# B&R Automation Studio project TD52 (part 15)

```c
/* Source: ctrttf.f */
#define ctrttf FORTRAN_WRAPPER(ctrttf)
extern void ctrttf(
    char   *transr,
    char   *uplo,
    ptrdiff_t *n,
    float  *a,
    ptrdiff_t *lda,
    float  *arf,
    ptrdiff_t *info
);

/* Source: ctrttp.f */
#define ctrttp FORTRAN_WRAPPER(ctrttp)
extern void ctrttp(
    char   *uplo,
    ptrdiff_t *n,
    float  *a,
    ptrdiff_t *lda,
    float  *ap,
    ptrdiff_t *info
);

/* Source: ctzrqf.f */
#define ctzrqf FORTRAN_WRAPPER(ctzrqf)
extern void ctzrqf(
    ptrdiff_t *m,
    ptrdiff_t *n,
    float  *a,
    ptrdiff_t *lda,
    float  *tau,
    ptrdiff_t *info
);

/* Source: ctzrzf.f */
#define ctzrzf FORTRAN_WRAPPER(ctzrzf)
extern void ctzrzf(
    ptrdiff_t *m,
    ptrdiff_t *n,
    float  *a,
    ptrdiff_t *lda,
    float  *tau,
    float  *work,
    ptrdiff_t *lwork,
    ptrdiff_t *info
);

/* Source: cung2l.f */
#define cung2l FORTRAN_WRAPPER(cung2l)
extern void cung2l(
    ptrdiff_t *m,
    ptrdiff_t *n,
    ptrdiff_t *k,
    float  *a,
    ptrdiff_t *lda,
    float  *tau,
    float  *work,
    ptrdiff_t *info
);

/* Source: cung2r.f */
#define cung2r FORTRAN_WRAPPER(cung2r)
extern void cung2r(
    ptrdiff_t *m,
    ptrdiff_t *n,
    ptrdiff_t *k,
    float  *a,
    ptrdiff_t *lda,
    float  *tau,
    float  *work,
    ptrdiff_t *info
);

/* Source: cungbr.f */
#define cungbr FORTRAN_WRAPPER(cungbr)
extern void cungbr(
    char   *vect,
    ptrdiff_t *m,
    ptrdiff_t *n,
    ptrdiff_t *k,
    float  *a,
    ptrdiff_t *lda,
    float  *tau,
    float  *work,
    ptrdiff_t *lwork,
    ptrdiff_t *info
);

/* Source: cunghr.f */
#define cunghr FORTRAN_WRAPPER(cunghr)
extern void cunghr(
    ptrdiff_t *n,
    ptrdiff_t *ilo,
    ptrdiff_t *ihi,
    float  *a,
    ptrdiff_t *lda,
    float  *tau,
    float  *work,
    ptrdiff_t *lwork,
    ptrdiff_t *info
);

/* Source: cungl2.f */
#define cungl2 FORTRAN_WRAPPER(cungl2)
extern void cungl2(
    ptrdiff_t *m,
    ptrdiff_t *n,
    ptrdiff_t *k,
    float  *a,
    ptrdiff_t *lda,
    float  *tau,
    float  *work,
    ptrdiff_t *info
);

/* Source: cunglq.f */
#define cunglq FORTRAN_WRAPPER(cunglq)
extern void cunglq(
    ptrdiff_t *m,
    ptrdiff_t *n,
    ptrdiff_t *k,
    float  *a,
    ptrdiff_t *lda,
    float  *tau,
    float  *work,
    ptrdiff_t *lwork,
    ptrdiff_t *info
);

/* Source: cungql.f */
#define cungql FORTRAN_WRAPPER(cungql)
extern void cungql(
    ptrdiff_t *m,
    ptrdiff_t *n,
    ptrdiff_t *k,
    float  *a,
    ptrdiff_t *lda,
    float  *tau,
    float  *work,
    ptrdiff_t *lwork,
    ptrdiff_t *info
);

/* Source: cungqr.f */
#define cungqr FORTRAN_WRAPPER(cungqr)
extern void cungqr(
    ptrdiff_t *m,
    ptrdiff_t *n,
    ptrdiff_t *k,
    float  *a,
    ptrdiff_t *lda,
    float  *tau,
    float  *work,
    ptrdiff_t *lwork,
    ptrdiff_t *info
);

/* Source: cungr2.f */
#define cungr2 FORTRAN_WRAPPER(cungr2)
extern void cungr2(
    ptrdiff_t *m,
    ptrdiff_t *n,
    ptrdiff_t *k,
    float  *a,
    ptrdiff_t *lda,
    float  *tau,
    float  *work,
    ptrdiff_t *info
);

/* Source: cungrq.f */
#define cungrq FORTRAN_WRAPPER(cungrq)
extern void cungrq(
    ptrdiff_t *m,
    ptrdiff_t *n,
    ptrdiff_t *k,
    float  *a,
    ptrdiff_t *lda,
    float  *tau,
    float  *work,
    ptrdiff_t *lwork,
    ptrdiff_t *info
);

/* Source: cungtr.f */
#define cungtr FORTRAN_WRAPPER(cungtr)
extern void cungtr(
    char   *uplo,
    ptrdiff_t *n,
    float  *a,
    ptrdiff_t *lda,
    float  *tau,
    float  *work,
    ptrdiff_t *lwork,
    ptrdiff_t *info
);

/* Source: cunm2l.f */
#define cunm2l FORTRAN_WRAPPER(cunm2l)
extern void cunm2l(
    char   *side,
    char   *trans,
    ptrdiff_t *m,
    ptrdiff_t *n,
    ptrdiff_t *k,
    float  *a,
    ptrdiff_t *lda,
    float  *tau,
    float  *c,
    ptrdiff_t *ldc,
    float  *work,
    ptrdiff_t *info
);

/* Source: cunm2r.f */
#define cunm2r FORTRAN_WRAPPER(cunm2r)
extern void cunm2r(
    char   *side,
    char   *trans,
    ptrdiff_t *m,
    ptrdiff_t *n,
    ptrdiff_t *k,
    float  *a,
    ptrdiff_t *lda,
    float  *tau,
    float  *c,
    ptrdiff_t *ldc,
    float  *work,
    ptrdiff_t *info
);

/* Source: cunmbr.f */
#define cunmbr FORTRAN_WRAPPER(cunmbr)
extern void cunmbr(
    char   *vect,
    char   *side,
    char   *trans,
    ptrdiff_t *m,
    ptrdiff_t *n,
    ptrdiff_t *k,
    float  *a,
    ptrdiff_t *lda,
    float  *tau,
    float  *c,
    ptrdiff_t *ldc,
    float  *work,
    ptrdiff_t *lwork,
    ptrdiff_t *info
);

/* Source: cunmhr.f */
#define cunmhr FORTRAN_WRAPPER(cunmhr)
extern void cunmhr(
    char   *side,
    char   *trans,
    ptrdiff_t *m,
    ptrdiff_t *n,
    ptrdiff_t *ilo,
    ptrdiff_t *ihi,
    float  *a,
    ptrdiff_t *lda,
    float  *tau,
    float  *c,
    ptrdiff_t *ldc,
    float  *work,
    ptrdiff_t *lwork,
    ptrdiff_t *info
);

/* Source: cunml2.f */
#define cunml2 FORTRAN_WRAPPER(cunml2)
extern void cunml2(
    char   *side,
    char   *trans,
    ptrdiff_t *m,
    ptrdiff_t *n,
    ptrdiff_t *k,
    float  *a,
    ptrdiff_t *lda,
    float  *tau,
    float  *c,
    ptrdiff_t *ldc,
    float  *work,
    ptrdiff_t *info
);

/* Source: cunmlq.f */
#define cunmlq FORTRAN_WRAPPER(cunmlq)
extern void cunmlq(
    char   *side,
    char   *trans,
    ptrdiff_t *m,
    ptrdiff_t *n,
    ptrdiff_t *k,
    float  *a,
    ptrdiff_t *lda,
    float  *tau,
    float  *c,
    ptrdiff_t *ldc,
    float  *work,
    ptrdiff_t *lwork,
    ptrdiff_t *info
);

/* Source: cunmql.f */
#define cunmql FORTRAN_WRAPPER(cunmql)
extern void cunmql(
    char   *side,
    char   *trans,
    ptrdiff_t *m,
    ptrdiff_t *n,
    ptrdiff_t *k,
    float  *a,
    ptrdiff_t *lda,
    float  *tau,
    float  *c,
    ptrdiff_t *ldc,
    float  *work,
    ptrdiff_t *lwork,
    ptrdiff_t *info
);

/* Source: cunmqr.f */
#define cunmqr FORTRAN_WRAPPER(cunmqr)
extern void cunmqr(
    char   *side,
    char   *trans,
    ptrdiff_t *m,
    ptrdiff_t *n,
    ptrdiff_t *k,
    float  *a,
    ptrdiff_t *lda,
    float  *tau,
    float  *c,
    ptrdiff_t *ldc,
    float  *work,
    ptrdiff_t *lwork,
    ptrdiff_t *info
);

/* Source: cunmr2.f */
#define cunmr2 FORTRAN_WRAPPER(cunmr2)
extern void cunmr2(
    char   *side,
    char   *trans,
    ptrdiff_t *m,
    ptrdiff_t *n,
    ptrdiff_t *k,
    float  *a,
    ptrdiff_t *lda,
    float  *tau,
    float  *c,
    ptrdiff_t *ldc,
    float  *work,
    ptrdiff_t *info
);

/* Source: cunmr3.f */
#define cunmr3 FORTRAN_WRAPPER(cunmr3)
extern void cunmr3(
    char   *side,
    char   *trans,
    ptrdiff_t *m,
    ptrdiff_t *n,
    ptrdiff_t *k,
    ptrdiff_t *l,
    float  *a,
    ptrdiff_t *lda,
    float  *tau,
    float  *c,
    ptrdiff_t *ldc,
    float  *work,
    ptrdiff_t *info
);

/* Source: cunmrq.f */
#define cunmrq FORTRAN_WRAPPER(cunmrq)
extern void cunmrq(
    char   *side,
    char   *trans,
    ptrdiff_t *m,
    ptrdiff_t *n,
    ptrdiff_t *k,
    float  *a,
    ptrdiff_t *lda,
    float  *tau,
    float  *c,
    ptrdiff_t *ldc,
    float  *work,
    ptrdiff_t *lwork,
    ptrdiff_t *info
);

/* Source: cunmrz.f */
#define cunmrz FORTRAN_WRAPPER(cunmrz)
extern void cunmrz(
    char   *side,
    char   *trans,
    ptrdiff_t *m,
    ptrdiff_t *n,
    ptrdiff_t *k,
    ptrdiff_t *l,
    float  *a,
    ptrdiff_t *lda,
    float  *tau,
    float  *c,
    ptrdiff_t *ldc,
    float  *work,
    ptrdiff_t *lwork,
    ptrdiff_t *info
);

/* Source: cunmtr.f */
#define cunmtr FORTRAN_WRAPPER(cunmtr)
extern void cunmtr(
    char   *side,
    char   *uplo,
    char   *trans,
    ptrdiff_t *m,
    ptrdiff_t *n,
    float  *a,
    ptrdiff_t *lda,
    float  *tau,
    float  *c,
    ptrdiff_t *ldc,
    float  *work,
    ptrdiff_t *lwork,
    ptrdiff_t *info
);

/* Source: cupgtr.f */
#define cupgtr FORTRAN_WRAPPER(cupgtr)
extern void cupgtr(
    char   *uplo,
    ptrdiff_t *n,
    float  *ap,
    float  *tau,
    float  *q,
    ptrdiff_t *ldq,
    float  *work,
    ptrdiff_t *info
);

/* Source: cupmtr.f */
#define cupmtr FORTRAN_WRAPPER(cupmtr)
extern void cupmtr(
    char   *side,
    char   *uplo,
    char   *trans,
    ptrdiff_t *m,
    ptrdiff_t *n,
    float  *ap,
    float  *tau,
    float  *c,
    ptrdiff_t *ldc,
    float  *work,
    ptrdiff_t *info
);

/* Source: dbdsdc.f */
#define dbdsdc FORTRAN_WRAPPER(dbdsdc)
extern void dbdsdc(
    char   *uplo,
    char   *compq,
    ptrdiff_t *n,
    double *d,
    double *e,
    double *u,
    ptrdiff_t *ldu,
    double *vt,
    ptrdiff_t *ldvt,
    double *q,
    ptrdiff_t *iq,
    double *work,
    ptrdiff_t *iwork,
    ptrdiff_t *info
);

/* Source: dbdsqr.f */
#define dbdsqr FORTRAN_WRAPPER(dbdsqr)
extern void dbdsqr(
    char   *uplo,
    ptrdiff_t *n,
    ptrdiff_t *ncvt,
    ptrdiff_t *nru,
    ptrdiff_t *ncc,
    double *d,
    double *e,
    double *vt,
    ptrdiff_t *ldvt,
    double *u,
    ptrdiff_t *ldu,
    double *c,
    ptrdiff_t *ldc,
    double *work,
    ptrdiff_t *info
);

/* Source: ddisna.f */
#define ddisna FORTRAN_WRAPPER(ddisna)
extern void ddisna(
    char   *job,
    ptrdiff_t *m,
    ptrdiff_t *n,
    double *d,
    double *sep,
    ptrdiff_t *info
);

/* Source: dgbbrd.f */
#define dgbbrd FORTRAN_WRAPPER(dgbbrd)
extern void dgbbrd(
    char   *vect,
    ptrdiff_t *m,
    ptrdiff_t *n,
    ptrdiff_t *ncc,
    ptrdiff_t *kl,
    ptrdiff_t *ku,
    double *ab,
    ptrdiff_t *ldab,
    double *d,
    double *e,
    double *q,
    ptrdiff_t *ldq,
    double *pt,
    ptrdiff_t *ldpt,
    double *c,
    ptrdiff_t *ldc,
    double *work,
    ptrdiff_t *info
);

/* Source: dgbcon.f */
#define dgbcon FORTRAN_WRAPPER(dgbcon)
extern void dgbcon(
    char   *norm,
    ptrdiff_t *n,
    ptrdiff_t *kl,
    ptrdiff_t *ku,
    double *ab,
    ptrdiff_t *ldab,
    ptrdiff_t *ipiv,
    double *anorm,
    double *rcond,
    double *work,
    ptrdiff_t *iwork,
    ptrdiff_t *info
);

/* Source: dgbequ.f */
#define dgbequ FORTRAN_WRAPPER(dgbequ)
extern void dgbequ(
    ptrdiff_t *m,
    ptrdiff_t *n,
    ptrdiff_t *kl,
    ptrdiff_t *ku,
    double *ab,
    ptrdiff_t *ldab,
    double *r,
    double *c,
    double *rowcnd,
    double *colcnd,
    double *amax,
    ptrdiff_t *info
);

/* Source: dgbequb.f */
#define dgbequb FORTRAN_WRAPPER(dgbequb)
extern void dgbequb(
    ptrdiff_t *m,
    ptrdiff_t *n,
    ptrdiff_t *kl,
    ptrdiff_t *ku,
    double *ab,
    ptrdiff_t *ldab,
    double *r,
    double *c,
    double *rowcnd,
    double *colcnd,
    double *amax,
    ptrdiff_t *info
);

/* Source: dgbrfs.f */
#define dgbrfs FORTRAN_WRAPPER(dgbrfs)
extern void dgbrfs(
    char   *trans,
    ptrdiff_t *n,
    ptrdiff_t *kl,
    ptrdiff_t *ku,
    ptrdiff_t *nrhs,
    double *ab,
    ptrdiff_t *ldab,
    double *afb,
    ptrdiff_t *ldafb,
    ptrdiff_t *ipiv,
    double *b,
    ptrdiff_t *ldb,
    double *x,
    ptrdiff_t *ldx,
    double *ferr,
    double *berr,
    double *work,
    ptrdiff_t *iwork,
    ptrdiff_t *info
);

/* Source: dgbsv.f */
#define dgbsv FORTRAN_WRAPPER(dgbsv)
extern void dgbsv(
    ptrdiff_t *n,
    ptrdiff_t *kl,
    ptrdiff_t *ku,
    ptrdiff_t *nrhs,
    double *ab,
    ptrdiff_t *ldab,
    ptrdiff_t *ipiv,
    double *b,
    ptrdiff_t *ldb,
    ptrdiff_t *info
);

/* Source: dgbsvx.f */
#define dgbsvx FORTRAN_WRAPPER(dgbsvx)
extern void dgbsvx(
    char   *fact,
    char   *trans,
    ptrdiff_t *n,
    ptrdiff_t *kl,
    ptrdiff_t *ku,
    ptrdiff_t *nrhs,
    double *ab,
    ptrdiff_t *ldab,
    double *afb,
    ptrdiff_t *ldafb,
    ptrdiff_t *ipiv,
    char   *equed,
    double *r,
    double *c,
    double *b,
    ptrdiff_t *ldb,
    double *x,
    ptrdiff_t *ldx,
    double *rcond,
    double *ferr,
    double *berr,
    double *work,
    ptrdiff_t *iwork,
    ptrdiff_t *info
);

/* Source: dgbtf2.f */
#define dgbtf2 FORTRAN_WRAPPER(dgbtf2)
extern void dgbtf2(
    ptrdiff_t *m,
    ptrdiff_t *n,
    ptrdiff_t *kl,
    ptrdiff_t *ku,
    double *ab,
    ptrdiff_t *ldab,
    ptrdiff_t *ipiv,
    ptrdiff_t *info
);

/* Source: dgbtrf.f */
#define dgbtrf FORTRAN_WRAPPER(dgbtrf)
extern void dgbtrf(
    ptrdiff_t *m,
    ptrdiff_t *n,
    ptrdiff_t *kl,
    ptrdiff_t *ku,
    double *ab,
    ptrdiff_t *ldab,
    ptrdiff_t *ipiv,
    ptrdiff_t *info
);

/* Source: dgbtrs.f */
#define dgbtrs FORTRAN_WRAPPER(dgbtrs)
extern void dgbtrs(
    char   *trans,
    ptrdiff_t *n,
    ptrdiff_t *kl,
    ptrdiff_t *ku,
    ptrdiff_t *nrhs,
    double *ab,
    ptrdiff_t *ldab,
    ptrdiff_t *ipiv,
    double *b,
    ptrdiff_t *ldb,
    ptrdiff_t *info
);

/* Source: dgebak.f */
#define dgebak FORTRAN_WRAPPER(dgebak)
extern void dgebak(
    char   *job,
    char   *side,
    ptrdiff_t *n,
    ptrdiff_t *ilo,
    ptrdiff_t *ihi,
    double *scale,
    ptrdiff_t *m,
    double *v,
    ptrdiff_t *ldv,
    ptrdiff_t *info
);

/* Source: dgebal.f */
#define dgebal FORTRAN_WRAPPER(dgebal)
extern void dgebal(
    char   *job,
    ptrdiff_t *n,
    double *a,
    ptrdiff_t *lda,
    ptrdiff_t *ilo,
    ptrdiff_t *ihi,
    double *scale,
    ptrdiff_t *info
);

/* Source: dgebd2.f */
#define dgebd2 FORTRAN_WRAPPER(dgebd2)
extern void dgebd2(
    ptrdiff_t *m,
    ptrdiff_t *n,
    double *a,
    ptrdiff_t *lda,
    double *d,
    double *e,
    double *tauq,
    double *taup,
    double *work,
    ptrdiff_t *info
);

/* Source: dgebrd.f */
#define dgebrd FORTRAN_WRAPPER(dgebrd)
extern void dgebrd(
    ptrdiff_t *m,
    ptrdiff_t *n,
    double *a,
    ptrdiff_t *lda,
    double *d,
    double *e,
    double *tauq,
    double *taup,
    double *work,
    ptrdiff_t *lwork,
    ptrdiff_t *info
);

/* Source: dgecon.f */
#define dgecon FORTRAN_WRAPPER(dgecon)
extern void dgecon(
    char   *norm,
    ptrdiff_t *n,
    double *a,
    ptrdiff_t *lda,
    double *anorm,
    double *rcond,
    double *work,
    ptrdiff_t *iwork,
    ptrdiff_t *info
);

/* Source: dgeequ.f */
#define dgeequ FORTRAN_WRAPPER(dgeequ)
extern void dgeequ(
    ptrdiff_t *m,
    ptrdiff_t *n,
    double *a,
    ptrdiff_t *lda,
    double *r,
    double *c,
    double *rowcnd,
    double *colcnd,
    double *amax,
    ptrdiff_t *info
);

/* Source: dgeequb.f */
#define dgeequb FORTRAN_WRAPPER(dgeequb)
extern void dgeequb(
    ptrdiff_t *m,
    ptrdiff_t *n,
    double *a,
    ptrdiff_t *lda,
    double *r,
    double *c,
    double *rowcnd,
    double *colcnd,
    double *amax,
    ptrdiff_t *info
);

/* Source: dgees.f */
#define dgees FORTRAN_WRAPPER(dgees)
extern void dgees(
    char   *jobvs,
    char   *sort,
    ptrdiff_t (*select)(),
    ptrdiff_t *n,
    double *a,
    ptrdiff_t *lda,
    ptrdiff_t *sdim,
    double *wr,
    double *wi,
    double *vs,
    ptrdiff_t *ldvs,
    double *work,
    ptrdiff_t *lwork,
    ptrdiff_t *bwork,
    ptrdiff_t *info
);

/* Source: dgeesx.f */
#define dgeesx FORTRAN_WRAPPER(dgeesx)
extern void dgeesx(
    char   *jobvs,
    char   *sort,
    ptrdiff_t (*select)(),
    char   *sense,
    ptrdiff_t *n,
    double *a,
    ptrdiff_t *lda,
    ptrdiff_t *sdim,
    double *wr,
    double *wi,
    double *vs,
    ptrdiff_t *ldvs,
    double *rconde,
    double *rcondv,
    double *work,
    ptrdiff_t *lwork,
    ptrdiff_t *iwork,
    ptrdiff_t *liwork,
    ptrdiff_t *bwork,
    ptrdiff_t *info
);

/* Source: dgeev.f */
#define dgeev FORTRAN_WRAPPER(dgeev)
extern void dgeev(
    char   *jobvl,
    char   *jobvr,
    ptrdiff_t *n,
    double *a,
    ptrdiff_t *lda,
    double *wr,
    double *wi,
    double *vl,
    ptrdiff_t *ldvl,
    double *vr,
    ptrdiff_t *ldvr,
    double *work,
    ptrdiff_t *lwork,
    ptrdiff_t *info
);

/* Source: dgeevx.f */
#define dgeevx FORTRAN_WRAPPER(dgeevx)
extern void dgeevx(
    char   *balanc,
    char   *jobvl,
    char   *jobvr,
    char   *sense,
    ptrdiff_t *n,
    double *a,
    ptrdiff_t *lda,
    double *wr,
    double *wi,
    double *vl,
    ptrdiff_t *ldvl,
    double *vr,
    ptrdiff_t *ldvr,
    ptrdiff_t *ilo,
    ptrdiff_t *ihi,
    double *scale,
    double *abnrm,
    double *rconde,
    double *rcondv,
    double *work,
    ptrdiff_t *lwork,
    ptrdiff_t *iwork,
    ptrdiff_t *info
);

/* Source: dgegs.f */
#define dgegs FORTRAN_WRAPPER(dgegs)
extern void dgegs(
    char   *jobvsl,
    char   *jobvsr,
    ptrdiff_t *n,
    double *a,
    ptrdiff_t *lda,
    double *b,
    ptrdiff_t *ldb,
    double *alphar,
    double *alphai,
    double *beta,
    double *vsl,
    ptrdiff_t *ldvsl,
    double *vsr,
    ptrdiff_t *ldvsr,
    double *work,
    ptrdiff_t *lwork,
    ptrdiff_t *info
);

/* Source: dgegv.f */
#define dgegv FORTRAN_WRAPPER(dgegv)
extern void dgegv(
    char   *jobvl,
    char   *jobvr,
    ptrdiff_t *n,
    double *a,
    ptrdiff_t *lda,
    double *b,
    ptrdiff_t *ldb,
    double *alphar,
    double *alphai,
    double *beta,
    double *vl,
    ptrdiff_t *ldvl,
    double *vr,
    ptrdiff_t *ldvr,
    double *work,
    ptrdiff_t *lwork,
    ptrdiff_t *info
);

/* Source: dgehd2.f */
#define dgehd2 FORTRAN_WRAPPER(dgehd2)
extern void dgehd2(
    ptrdiff_t *n,
    ptrdiff_t *ilo,
    ptrdiff_t *ihi,
    double *a,
    ptrdiff_t *lda,
    double *tau,
    double *work,
    ptrdiff_t *info
);

/* Source: dgehrd.f */
#define dgehrd FORTRAN_WRAPPER(dgehrd)
extern void dgehrd(
    ptrdiff_t *n,
    ptrdiff_t *ilo,
    ptrdiff_t *ihi,
    double *a,
    ptrdiff_t *lda,
    double *tau,
    double *work,
    ptrdiff_t *lwork,
    ptrdiff_t *info
);

/* Source: dgejsv.f */
#define dgejsv FORTRAN_WRAPPER(dgejsv)
extern void dgejsv(
    char   *joba,
    char   *jobu,
    char   *jobv,
    char   *jobr,
    char   *jobt,
    char   *jobp,
    ptrdiff_t *m,
    ptrdiff_t *n,
    double *a,
    ptrdiff_t *lda,
    double *sva,
    double *u,
    ptrdiff_t *ldu,
    double *v,
    ptrdiff_t *ldv,
    double *work,
    ptrdiff_t *lwork,
    ptrdiff_t *iwork,
    ptrdiff_t *info
);

/* Source: dgelq2.f */
#define dgelq2 FORTRAN_WRAPPER(dgelq2)
extern void dgelq2(
    ptrdiff_t *m,
    ptrdiff_t *n,
    double *a,
    ptrdiff_t *lda,
    double *tau,
    double *work,
    ptrdiff_t *info
);

/* Source: dgelqf.f */
#define dgelqf FORTRAN_WRAPPER(dgelqf)
extern void dgelqf(
    ptrdiff_t *m,
    ptrdiff_t *n,
    double *a,
    ptrdiff_t *lda,
    double *tau,
    double *work,
    ptrdiff_t *lwork,
    ptrdiff_t *info
);

/* Source: dgels.f */
#define dgels FORTRAN_WRAPPER(dgels)
extern void dgels(
    char   *trans,
    ptrdiff_t *m,
    ptrdiff_t *n,
    ptrdiff_t *nrhs,
    double *a,
    ptrdiff_t *lda,
    double *b,
    ptrdiff_t *ldb,
    double *work,
    ptrdiff_t *lwork,
    ptrdiff_t *info
);

/* Source: dgelsd.f */
#define dgelsd FORTRAN_WRAPPER(dgelsd)
extern void dgelsd(
    ptrdiff_t *m,
    ptrdiff_t *n,
    ptrdiff_t *nrhs,
    double *a,
    ptrdiff_t *lda,
    double *b,
    ptrdiff_t *ldb,
    double *s,
    double *rcond,
    ptrdiff_t *rank,
    double *work,
    ptrdiff_t *lwork,
    ptrdiff_t *iwork,
    ptrdiff_t *info
);

/* Source: dgelss.f */
#define dgelss FORTRAN_WRAPPER(dgelss)
extern void dgelss(
    ptrdiff_t *m,
    ptrdiff_t *n,
    ptrdiff_t *nrhs,
    double *a,
    ptrdiff_t *lda,
    double *b,
    ptrdiff_t *ldb,
    double *s,
    double *rcond,
    ptrdiff_t *rank,
    double *work,
    ptrdiff_t *lwork,
    ptrdiff_t *info
);

/* Source: dgelsx.f */
#define dgelsx FORTRAN_WRAPPER(dgelsx)
extern void dgelsx(
    ptrdiff_t *m,
    ptrdiff_t *n,
    ptrdiff_t *nrhs,
    double *a,
    ptrdiff_t *lda,
    double *b,
    ptrdiff_t *ldb,
    ptrdiff_t *jpvt,
    double *rcond,
    ptrdiff_t *rank,
    double *work,
    ptrdiff_t *info
);

/* Source: dgelsy.f */
#define dgelsy FORTRAN_WRAPPER(dgelsy)
extern void dgelsy(
    ptrdiff_t *m,
    ptrdiff_t *n,
    ptrdiff_t *nrhs,
    double *a,
    ptrdiff_t *lda,
    double *b,
    ptrdiff_t *ldb,
    ptrdiff_t *jpvt,
    double *rcond,
    ptrdiff_t *rank,
    double *work,
    ptrdiff_t *lwork,
    ptrdiff_t *info
);

/* Source: dgeql2.f */
#define dgeql2 FORTRAN_WRAPPER(dgeql2)
extern void dgeql2(
    ptrdiff_t *m,
    ptrdiff_t *n,
    double *a,
    ptrdiff_t *lda,
    double *tau,
    double *work,
    ptrdiff_t *info
);

/* Source: dgeqlf.f */
#define dgeqlf FORTRAN_WRAPPER(dgeqlf)
extern void dgeqlf(
    ptrdiff_t *m,
    ptrdiff_t *n,
    double *a,
    ptrdiff_t *lda,
    double *tau,
    double *work,
    ptrdiff_t *lwork,
    ptrdiff_t *info
);

/* Source: dgeqp3.f */
#define dgeqp3 FORTRAN_WRAPPER(dgeqp3)
extern void dgeqp3(
    ptrdiff_t *m,
    ptrdiff_t *n,
    double *a,
    ptrdiff_t *lda,
    ptrdiff_t *jpvt,
    double *tau,
    double *work,
    ptrdiff_t *lwork,
    ptrdiff_t *info
);

/* Source: dgeqpf.f */
#define dgeqpf FORTRAN_WRAPPER(dgeqpf)
extern void dgeqpf(
    ptrdiff_t *m,
    ptrdiff_t *n,
    double *a,
    ptrdiff_t *lda,
    ptrdiff_t *jpvt,
    double *tau,
    double *work,
    ptrdiff_t *info
);

/* Source: dgeqr2.f */
#define dgeqr2 FORTRAN_WRAPPER(dgeqr2)
extern void dgeqr2(
    ptrdiff_t *m,
    ptrdiff_t *n,
    double *a,
    ptrdiff_t *lda,
    double *tau,
    double *work,
    ptrdiff_t *info
);

/* Source: dgeqr2p.f */
#define dgeqr2p FORTRAN_WRAPPER(dgeqr2p)
extern void dgeqr2p(
    ptrdiff_t *m,
    ptrdiff_t *n,
    double *a,
    ptrdiff_t *lda,
    double *tau,
    double *work,
    ptrdiff_t *info
);

/* Source: dgeqrf.f */
#define dgeqrf FORTRAN_WRAPPER(dgeqrf)
extern void dgeqrf(
    ptrdiff_t *m,
    ptrdiff_t *n,
    double *a,
    ptrdiff_t *lda,
    double *tau,
    double *work,
    ptrdiff_t *lwork,
    ptrdiff_t *info
);

/* Source: dgeqrfp.f */
#define dgeqrfp FORTRAN_WRAPPER(dgeqrfp)
extern void dgeqrfp(
    ptrdiff_t *m,
    ptrdiff_t *n,
    double *a,
    ptrdiff_t *lda,
    double *tau,
    double *work,
    ptrdiff_t *lwork,
    ptrdiff_t *info
);

/* Source: dgerfs.f */
#define dgerfs FORTRAN_WRAPPER(dgerfs)
extern void dgerfs(
    char   *trans,
    ptrdiff_t *n,
    ptrdiff_t *nrhs,
    double *a,
    ptrdiff_t *lda,
    double *af,
    ptrdiff_t *ldaf,
    ptrdiff_t *ipiv,
    double *b,
    ptrdiff_t *ldb,
    double *x,
    ptrdiff_t *ldx,
    double *ferr,
    double *berr,
    double *work,
    ptrdiff_t *iwork,
    ptrdiff_t *info
);

/* Source: dgerq2.f */
#define dgerq2 FORTRAN_WRAPPER(dgerq2)
extern void dgerq2(
    ptrdiff_t *m,
    ptrdiff_t *n,
    double *a,
    ptrdiff_t *lda,
    double *tau,
    double *work,
    ptrdiff_t *info
);

/* Source: dgerqf.f */
#define dgerqf FORTRAN_WRAPPER(dgerqf)
extern void dgerqf(
    ptrdiff_t *m,
    ptrdiff_t *n,
    double *a,
    ptrdiff_t *lda,
    double *tau,
    double *work,
    ptrdiff_t *lwork,
    ptrdiff_t *info
);

/* Source: dgesc2.f */
#define dgesc2 FORTRAN_WRAPPER(dgesc2)
extern void dgesc2(
    ptrdiff_t *n,
    double *a,
    ptrdiff_t *lda,
    double *rhs,
    ptrdiff_t *ipiv,
    ptrdiff_t *jpiv,
    double *scale
);

/* Source: dgesdd.f */
#define dgesdd FORTRAN_WRAPPER(dgesdd)
extern void dgesdd(
    char   *jobz,
    ptrdiff_t *m,
    ptrdiff_t *n,
    double *a,
    ptrdiff_t *lda,
    double *s,
    double *u,
    ptrdiff_t *ldu,
    double *vt,
    ptrdiff_t *ldvt,
    double *work,
    ptrdiff_t *lwork,
    ptrdiff_t *iwork,
    ptrdiff_t *info
);

/* Source: dgesv.f */
#define dgesv FORTRAN_WRAPPER(dgesv)
extern void dgesv(
    ptrdiff_t *n,
    ptrdiff_t *nrhs,
    double *a,
    ptrdiff_t *lda,
    ptrdiff_t *ipiv,
    double *b,
    ptrdiff_t *ldb,
    ptrdiff_t *info
);

/* Source: dgesvd.f */
#define dgesvd FORTRAN_WRAPPER(dgesvd)
extern void dgesvd(
    char   *jobu,
    char   *jobvt,
    ptrdiff_t *m,
    ptrdiff_t *n,
    double *a,
    ptrdiff_t *lda,
    double *s,
    double *u,
    ptrdiff_t *ldu,
    double *vt,
    ptrdiff_t *ldvt,
    double *work,
    ptrdiff_t *lwork,
    ptrdiff_t *info
);

/* Source: dgesvj.f */
#define dgesvj FORTRAN_WRAPPER(dgesvj)
extern void dgesvj(
    char   *joba,
    char   *jobu,
    char   *jobv,
    ptrdiff_t *m,
    ptrdiff_t *n,
    double *a,
    ptrdiff_t *lda,
    double *sva,
    ptrdiff_t *mv,
    double *v,
    ptrdiff_t *ldv,
    double *work,
    ptrdiff_t *lwork,
    ptrdiff_t *info
);

/* Source: dgesvx.f */
#define dgesvx FORTRAN_WRAPPER(dgesvx)
extern void dgesvx(
    char   *fact,
    char   *trans,
    ptrdiff_t *n,
    ptrdiff_t *nrhs,
    double *a,
    ptrdiff_t *lda,
    double *af,
    ptrdiff_t *ldaf,
    ptrdiff_t *ipiv,
    char   *equed,
    double *r,
    double *c,
    double *b,
    ptrdiff_t *ldb,
    double *x,
    ptrdiff_t *ldx,
    double *rcond,
    double *ferr,
    double *berr,
    double *work,
    ptrdiff_t *iwork,
    ptrdiff_t *info
);

/* Source: dgetc2.f */
#define dgetc2 FORTRAN_WRAPPER(dgetc2)
extern void dgetc2(
    ptrdiff_t *n,
    double *a,
    ptrdiff_t *lda,
    ptrdiff_t *ipiv,
    ptrdiff_t *jpiv,
    ptrdiff_t *info
);

/* Source: dgetf2.f */
#define dgetf2 FORTRAN_WRAPPER(dgetf2)
extern void dgetf2(
    ptrdiff_t *m,
    ptrdiff_t *n,
    double *a,
    ptrdiff_t *lda,
    ptrdiff_t *ipiv,
    ptrdiff_t *info
);

/* Source: dgetrf.f */
#define dgetrf FORTRAN_WRAPPER(dgetrf)
extern void dgetrf(
    ptrdiff_t *m,
    ptrdiff_t *n,
    double *a,
    ptrdiff_t *lda,
    ptrdiff_t *ipiv,
    ptrdiff_t *info
);

/* Source: dgetri.f */
#define dgetri FORTRAN_WRAPPER(dgetri)
extern void dgetri(
    ptrdiff_t *n,
    double *a,
    ptrdiff_t *lda,
    ptrdiff_t *ipiv,
    double *work,
    ptrdiff_t *lwork,
    ptrdiff_t *info
);

/* Source: dgetrs.f */
#define dgetrs FORTRAN_WRAPPER(dgetrs)
extern void dgetrs(
    char   *trans,
    ptrdiff_t *n,
    ptrdiff_t *nrhs,
    double *a,
    ptrdiff_t *lda,
    ptrdiff_t *ipiv,
    double *b,
    ptrdiff_t *ldb,
    ptrdiff_t *info
);

/* Source: dggbak.f */
#define dggbak FORTRAN_WRAPPER(dggbak)
extern void dggbak(
    char   *job,
    char   *side,
    ptrdiff_t *n,
    ptrdiff_t *ilo,
    ptrdiff_t *ihi,
    double *lscale,
    double *rscale,
    ptrdiff_t *m,
    double *v,
    ptrdiff_t *ldv,
    ptrdiff_t *info
);

/* Source: dggbal.f */
#define dggbal FORTRAN_WRAPPER(dggbal)
extern void dggbal(
    char   *job,
    ptrdiff_t *n,
    double *a,
    ptrdiff_t *lda,
    double *b,
    ptrdiff_t *ldb,
    ptrdiff_t *ilo,
    ptrdiff_t *ihi,
    double *lscale,
    double *rscale,
    double *work,
    ptrdiff_t *info
);

/* Source: dgges.f */
#define dgges FORTRAN_WRAPPER(dgges)
extern void dgges(
    char   *jobvsl,
    char   *jobvsr,
    char   *sort,
    ptrdiff_t (*selctg)(),
    ptrdiff_t *n,
    double *a,
    ptrdiff_t *lda,
    double *b,
    ptrdiff_t *ldb,
    ptrdiff_t *sdim,
    double *alphar,
    double *alphai,
    double *beta,
    double *vsl,
    ptrdiff_t *ldvsl,
    double *vsr,
    ptrdiff_t *ldvsr,
    double *work,
    ptrdiff_t *lwork,
    ptrdiff_t *bwork,
    ptrdiff_t *info
);

/* Source: dggesx.f */
#define dggesx FORTRAN_WRAPPER(dggesx)
extern void dggesx(
    char   *jobvsl,
    char   *jobvsr,
    char   *sort,
    ptrdiff_t (*selctg)(),
    char   *sense,
    ptrdiff_t *n,
    double *a,
    ptrdiff_t *lda,
    double *b,
    ptrdiff_t *ldb,
    ptrdiff_t *sdim,
    double *alphar,
    double *alphai,
    double *beta,
    double *vsl,
    ptrdiff_t *ldvsl,
    double *vsr,
    ptrdiff_t *ldvsr,
    double *rconde,
    double *rcondv,
    double *work,
    ptrdiff_t *lwork,
    ptrdiff_t *iwork,
    ptrdiff_t *liwork,
    ptrdiff_t *bwork,
    ptrdiff_t *info
);

/* Source: dggev.f */
#define dggev FORTRAN_WRAPPER(dggev)
extern void dggev(
    char   *jobvl,
    char   *jobvr,
    ptrdiff_t *n,
    double *a,
    ptrdiff_t *lda,
    double *b,
    ptrdiff_t *ldb,
    double *alphar,
    double *alphai,
    double *beta,
    double *vl,
    ptrdiff_t *ldvl,
    double *vr,
    ptrdiff_t *ldvr,
    double *work,
    ptrdiff_t *lwork,
    ptrdiff_t *info
);

/* Source: dggevx.f */
#define dggevx FORTRAN_WRAPPER(dggevx)
extern void dggevx(
    char   *balanc,
    char   *jobvl,
    char   *jobvr,
    char   *sense,
    ptrdiff_t *n,
    double *a,
    ptrdiff_t *lda,
    double *b,
    ptrdiff_t *ldb,
    double *alphar,
    double *alphai,
    double *beta,
    double *vl,
    ptrdiff_t *ldvl,
    double *vr,
    ptrdiff_t *ldvr,
    ptrdiff_t *ilo,
    ptrdiff_t *ihi,
    double *lscale,
    double *rscale,
    double *abnrm,
    double *bbnrm,
    double *rconde,
    double *rcondv,
    double *work,
    ptrdiff_t *lwork,
    ptrdiff_t *iwork,
    ptrdiff_t *bwork,
    ptrdiff_t *info
);

/* Source: dggglm.f */
#define dggglm FORTRAN_WRAPPER(dggglm)
extern void dggglm(
    ptrdiff_t *n,
    ptrdiff_t *m,
    ptrdiff_t *p,
    double *a,
    ptrdiff_t *lda,
    double *b,
    ptrdiff_t *ldb,
    double *d,
    double *x,
    double *y,
    double *work,
    ptrdiff_t *lwork,
    ptrdiff_t *info
);

/* Source: dgghrd.f */
#define dgghrd FORTRAN_WRAPPER(dgghrd)
extern void dgghrd(
    char   *compq,
    char   *compz,
    ptrdiff_t *n,
    ptrdiff_t *ilo,
    ptrdiff_t *ihi,
    double *a,
    ptrdiff_t *lda,
    double *b,
    ptrdiff_t *ldb,
    double *q,
    ptrdiff_t *ldq,
    double *z,
    ptrdiff_t *ldz,
    ptrdiff_t *info
);

/* Source: dgglse.f */
#define dgglse FORTRAN_WRAPPER(dgglse)
extern void dgglse(
    ptrdiff_t *m,
    ptrdiff_t *n,
    ptrdiff_t *p,
    double *a,
    ptrdiff_t *lda,
    double *b,
    ptrdiff_t *ldb,
    double *c,
    double *d,
    double *x,
    double *work,
    ptrdiff_t *lwork,
    ptrdiff_t *info
);

/* Source: dggqrf.f */
#define dggqrf FORTRAN_WRAPPER(dggqrf)
extern void dggqrf(
    ptrdiff_t *n,
    ptrdiff_t *m,
    ptrdiff_t *p,
    double *a,
    ptrdiff_t *lda,
    double *taua,
    double *b,
    ptrdiff_t *ldb,
    double *taub,
    double *work,
    ptrdiff_t *lwork,
    ptrdiff_t *info
);

/* Source: dggrqf.f */
#define dggrqf FORTRAN_WRAPPER(dggrqf)
extern void dggrqf(
    ptrdiff_t *m,
    ptrdiff_t *p,
    ptrdiff_t *n,
    double *a,
    ptrdiff_t *lda,
    double *taua,
    double *b,
    ptrdiff_t *ldb,
    double *taub,
    double *work,
    ptrdiff_t *lwork,
    ptrdiff_t *info
);

/* Source: dggsvd.f */
#define dggsvd FORTRAN_WRAPPER(dggsvd)
extern void dggsvd(
    char   *jobu,
    char   *jobv,
    char   *jobq,
    ptrdiff_t *m,
    ptrdiff_t *n,
    ptrdiff_t *p,
    ptrdiff_t *k,
    ptrdiff_t *l,
    double *a,
    ptrdiff_t *lda,
    double *b,
    ptrdiff_t *ldb,
    double *alpha,
    double *beta,
    double *u,
    ptrdiff_t *ldu,
    double *v,
    ptrdiff_t *ldv,
    double *q,
    ptrdiff_t *ldq,
    double *work,
    ptrdiff_t *iwork,
    ptrdiff_t *info
);

/* Source: dggsvp.f */
#define dggsvp FORTRAN_WRAPPER(dggsvp)
extern void dggsvp(
    char   *jobu,
    char   *jobv,
    char   *jobq,
    ptrdiff_t *m,
    ptrdiff_t *p,
    ptrdiff_t *n,
    double *a,
    ptrdiff_t *lda,
    double *b,
    ptrdiff_t *ldb,
    double *tola,
    double *tolb,
    ptrdiff_t *k,
    ptrdiff_t *l,
    double *u,
    ptrdiff_t *ldu,
    double *v,
    ptrdiff_t *ldv,
    double *q,
    ptrdiff_t *ldq,
    ptrdiff_t *iwork,
    double *tau,
    double *work,
    ptrdiff_t *info
);

/* Source: dgsvj0.f */
#define dgsvj0 FORTRAN_WRAPPER(dgsvj0)
extern void dgsvj0(
    char   *jobv,
    ptrdiff_t *m,
    ptrdiff_t *n,
    double *a,
    ptrdiff_t *lda,
    double *d,
    double *sva,
    ptrdiff_t *mv,
    double *v,
    ptrdiff_t *ldv,
    double *eps,
    double *sfmin,
    double *tol,
    ptrdiff_t *nsweep,
    double *work,
    ptrdiff_t *lwork,
    ptrdiff_t *info
);

/* Source: dgsvj1.f */
#define dgsvj1 FORTRAN_WRAPPER(dgsvj1)
extern void dgsvj1(
    char   *jobv,
    ptrdiff_t *m,
    ptrdiff_t *n,
    ptrdiff_t *n1,
    double *a,
    ptrdiff_t *lda,
    double *d,
    double *sva,
    ptrdiff_t *mv,
    double *v,
    ptrdiff_t *ldv,
    double *eps,
    double *sfmin,
    double *tol,
    ptrdiff_t *nsweep,
    double *work,
    ptrdiff_t *lwork,
    ptrdiff_t *info
);

/* Source: dgtcon.f */
#define dgtcon FORTRAN_WRAPPER(dgtcon)
extern void dgtcon(
    char   *norm,
    ptrdiff_t *n,
    double *dl,
    double *d,
    double *du,
    double *du2,
    ptrdiff_t *ipiv,
    double *anorm,
    double *rcond,
    double *work,
    ptrdiff_t *iwork,
    ptrdiff_t *info
);

/* Source: dgtrfs.f */
#define dgtrfs FORTRAN_WRAPPER(dgtrfs)
extern void dgtrfs(
    char   *trans,
    ptrdiff_t *n,
    ptrdiff_t *nrhs,
    double *dl,
    double *d,
    double *du,
    double *dlf,
    double *df,
    double *duf,
    double *du2,
    ptrdiff_t *ipiv,
    double *b,
    ptrdiff_t *ldb,
    double *x,
    ptrdiff_t *ldx,
    double *ferr,
    double *berr,
    double *work,
    ptrdiff_t *iwork,
    ptrdiff_t *info
);

/* Source: dgtsv.f */
#define dgtsv FORTRAN_WRAPPER(dgtsv)
extern void dgtsv(
    ptrdiff_t *n,
    ptrdiff_t *nrhs,
    double *dl,
    double *d,
    double *du,
    double *b,
    ptrdiff_t *ldb,
    ptrdiff_t *info
);

/* Source: dgtsvx.f */
#define dgtsvx FORTRAN_WRAPPER(dgtsvx)
extern void dgtsvx(
    char   *fact,
    char   *trans,
    ptrdiff_t *n,
    ptrdiff_t *nrhs,
    double *dl,
    double *d,
    double *du,
    double *dlf,
    double *df,
    double *duf,
    double *du2,
    ptrdiff_t *ipiv,
    double *b,
    ptrdiff_t *ldb,
    double *x,
    ptrdiff_t *ldx,
    double *rcond,
    double *ferr,
    double *berr,
    double *work,
    ptrdiff_t *iwork,
    ptrdiff_t *info
);

/* Source: dgttrf.f */
#define dgttrf FORTRAN_WRAPPER(dgttrf)
extern void dgttrf(
    ptrdiff_t *n,
    double *dl,
    double *d,
    double *du,
    double *du2,
    ptrdiff_t *ipiv,
    ptrdiff_t *info
);

/* Source: dgttrs.f */
#define dgttrs FORTRAN_WRAPPER(dgttrs)
extern void dgttrs(
    char   *trans,
    ptrdiff_t *n,
    ptrdiff_t *nrhs,
    double *dl,
    double *d,
    double *du,
    double *du2,
    ptrdiff_t *ipiv,
    double *b,
    ptrdiff_t *ldb,
    ptrdiff_t *info
);

/* Source: dgtts2.f */
#define dgtts2 FORTRAN_WRAPPER(dgtts2)
extern void dgtts2(
    ptrdiff_t *itrans,
    ptrdiff_t *n,
    ptrdiff_t *nrhs,
    double *dl,
    double *d,
    double *du,
    double *du2,
    ptrdiff_t *ipiv,
    double *b,
    ptrdiff_t *ldb
);

/* Source: dhgeqz.f */
#define dhgeqz FORTRAN_WRAPPER(dhgeqz)
extern void dhgeqz(
    char   *job,
    char   *compq,
    char   *compz,
    ptrdiff_t *n,
    ptrdiff_t *ilo,
    ptrdiff_t *ihi,
    double *h,
    ptrdiff_t *ldh,
    double *t,
    ptrdiff_t *ldt,
    double *alphar,
    double *alphai,
    double *beta,
    double *q,
    ptrdiff_t *ldq,
    double *z,
    ptrdiff_t *ldz,
    double *work,
    ptrdiff_t *lwork,
    ptrdiff_t *info
);

/* Source: dhsein.f */
#define dhsein FORTRAN_WRAPPER(dhsein)
extern void dhsein(
    char   *side,
    char   *eigsrc,
    char   *initv,
    ptrdiff_t *select,
    ptrdiff_t *n,
    double *h,
    ptrdiff_t *ldh,
    double *wr,
    double *wi,
    double *vl,
    ptrdiff_t *ldvl,
    double *vr,
    ptrdiff_t *ldvr,
    ptrdiff_t *mm,
    ptrdiff_t *m,
    double *work,
    ptrdiff_t *ifaill,
    ptrdiff_t *ifailr,
    ptrdiff_t *info
);

/* Source: dhseqr.f */
#define dhseqr FORTRAN_WRAPPER(dhseqr)
extern void dhseqr(
    char   *job,
    char   *compz,
    ptrdiff_t *n,
    ptrdiff_t *ilo,
    ptrdiff_t *ihi,
    double *h,
    ptrdiff_t *ldh,
    double *wr,
    double *wi,
    double *z,
    ptrdiff_t *ldz,
    double *work,
    ptrdiff_t *lwork,
    ptrdiff_t *info
);

/* Source: disnan.f */
#define disnan FORTRAN_WRAPPER(disnan)
extern ptrdiff_t disnan(
    double *din
);

/* Source: dlabad.f */
#define dlabad FORTRAN_WRAPPER(dlabad)
extern void dlabad(
    double *small,
    double *large
);

/* Source: dlabrd.f */
#define dlabrd FORTRAN_WRAPPER(dlabrd)
extern void dlabrd(
    ptrdiff_t *m,
    ptrdiff_t *n,
    ptrdiff_t *nb,
    double *a,
    ptrdiff_t *lda,
    double *d,
    double *e,
    double *tauq,
    double *taup,
    double *x,
    ptrdiff_t *ldx,
    double *y,
    ptrdiff_t *ldy
);

/* Source: dlacn2.f */
#define dlacn2 FORTRAN_WRAPPER(dlacn2)
extern void dlacn2(
    ptrdiff_t *n,
    double *v,
    double *x,
    ptrdiff_t *isgn,
    double *est,
    ptrdiff_t *kase,
    ptrdiff_t *isave
);

/* Source: dlacon.f */
#define dlacon FORTRAN_WRAPPER(dlacon)
extern void dlacon(
    ptrdiff_t *n,
    double *v,
    double *x,
    ptrdiff_t *isgn,
    double *est,
    ptrdiff_t *kase
);

/* Source: dlacpy.f */
#define dlacpy FORTRAN_WRAPPER(dlacpy)
extern void dlacpy(
    char   *uplo,
    ptrdiff_t *m,
    ptrdiff_t *n,
    double *a,
    ptrdiff_t *lda,
    double *b,
    ptrdiff_t *ldb
);

/* Source: dladiv.f */
#define dladiv FORTRAN_WRAPPER(dladiv)
extern void dladiv(
    double *a,
    double *b,
    double *c,
    double *d,
    double *p,
    double *q
);

/* Source: dlae2.f */
#define dlae2 FORTRAN_WRAPPER(dlae2)
extern void dlae2(
    double *a,
    double *b,
    double *c,
    double *rt1,
    double *rt2
);

/* Source: dlaebz.f */
#define dlaebz FORTRAN_WRAPPER(dlaebz)
extern void dlaebz(
    ptrdiff_t *ijob,
    ptrdiff_t *nitmax,
    ptrdiff_t *n,
    ptrdiff_t *mmax,
    ptrdiff_t *minp,
    ptrdiff_t *nbmin,
    double *abstol,
    double *reltol,
    double *pivmin,
    double *d,
    double *e,
    double *e2,
    ptrdiff_t *nval,
    double *ab,
    double *c,
    ptrdiff_t *mout,
    ptrdiff_t *nab,
    double *work,
    ptrdiff_t *iwork,
    ptrdiff_t *info
);

/* Source: dlaed0.f */
#define dlaed0 FORTRAN_WRAPPER(dlaed0)
extern void dlaed0(
    ptrdiff_t *icompq,
    ptrdiff_t *qsiz,
    ptrdiff_t *n,
    double *d,
    double *e,
    double *q,
    ptrdiff_t *ldq,
    double *qstore,
    ptrdiff_t *ldqs,
    double *work,
    ptrdiff_t *iwork,
    ptrdiff_t *info
);

/* Source: dlaed1.f */
#define dlaed1 FORTRAN_WRAPPER(dlaed1)
extern void dlaed1(
    ptrdiff_t *n,
    double *d,
    double *q,
    ptrdiff_t *ldq,
    ptrdiff_t *indxq,
    double *rho,
    ptrdiff_t *cutpnt,
    double *work,
    ptrdiff_t *iwork,
    ptrdiff_t *info
);

/* Source: dlaed2.f */
#define dlaed2 FORTRAN_WRAPPER(dlaed2)
extern void dlaed2(
    ptrdiff_t *k,
    ptrdiff_t *n,
    ptrdiff_t *n1,
    double *d,
    double *q,
    ptrdiff_t *ldq,
    ptrdiff_t *indxq,
    double *rho,
    double *z,
    double *dlamda,
    double *w,
    double *q2,
    ptrdiff_t *indx,
    ptrdiff_t *indxc,
    ptrdiff_t *indxp,
    ptrdiff_t *coltyp,
    ptrdiff_t *info
);

/* Source: dlaed3.f */
#define dlaed3 FORTRAN_WRAPPER(dlaed3)
extern void dlaed3(
    ptrdiff_t *k,
    ptrdiff_t *n,
    ptrdiff_t *n1,
    double *d,
    double *q,
    ptrdiff_t *ldq,
    double *rho,
    double *dlamda,
    double *q2,
    ptrdiff_t *indx,
    ptrdiff_t *ctot,
    double *w,
    double *s,
    ptrdiff_t *info
);

/* Source: dlaed4.f */
#define dlaed4 FORTRAN_WRAPPER(dlaed4)
extern void dlaed4(
    ptrdiff_t *n,
    ptrdiff_t *i,
    double *d,
    double *z,
    double *delta,
    double *rho,
    double *dlam,
    ptrdiff_t *info
);

/* Source: dlaed5.f */
#define dlaed5 FORTRAN_WRAPPER(dlaed5)
extern void dlaed5(
    ptrdiff_t *i,
    double *d,
    double *z,
    double *delta,
    double *rho,
    double *dlam
);

/* Source: dlaed6.f */
#define dlaed6 FORTRAN_WRAPPER(dlaed6)
extern void dlaed6(
    ptrdiff_t *kniter,
    ptrdiff_t *orgati,
    double *rho,
    double *d,
    double *z,
    double *finit,
    double *tau,
    ptrdiff_t *info
);

/* Source: dlaed7.f */
#define dlaed7 FORTRAN_WRAPPER(dlaed7)
extern void dlaed7(
    ptrdiff_t *icompq,
    ptrdiff_t *n,
    ptrdiff_t *qsiz,
    ptrdiff_t *tlvls,
    ptrdiff_t *curlvl,
    ptrdiff_t *curpbm,
    double *d,
    double *q,
    ptrdiff_t *ldq,
    ptrdiff_t *indxq,
    double *rho,
    ptrdiff_t *cutpnt,
    double *qstore,
    ptrdiff_t *qptr,
    ptrdiff_t *prmptr,
    ptrdiff_t *perm,
    ptrdiff_t *givptr,
    ptrdiff_t *givcol,
    double *givnum,
    double *work,
    ptrdiff_t *iwork,
    ptrdiff_t *info
);

/* Source: dlaed8.f */
#define dlaed8 FORTRAN_WRAPPER(dlaed8)
extern void dlaed8(
    ptrdiff_t *icompq,
    ptrdiff_t *k,
    ptrdiff_t *n,
    ptrdiff_t *qsiz,
    double *d,
    double *q,
    ptrdiff_t *ldq,
    ptrdiff_t *indxq,
    double *rho,
    ptrdiff_t *cutpnt,
    double *z,
    double *dlamda,
    double *q2,
    ptrdiff_t *ldq2,
    double *w,
    ptrdiff_t *perm,
    ptrdiff_t *givptr,
    ptrdiff_t *givcol,
    double *givnum,
    ptrdiff_t *indxp,
    ptrdiff_t *indx,
    ptrdiff_t *info
);

/* Source: dlaed9.f */
#define dlaed9 FORTRAN_WRAPPER(dlaed9)
extern void dlaed9(
    ptrdiff_t *k,
    ptrdiff_t *kstart,
    ptrdiff_t *kstop,
    ptrdiff_t *n,
    double *d,
    double *q,
    ptrdiff_t *ldq,
    double *rho,
    double *dlamda,
    double *w,
    double *s,
    ptrdiff_t *lds,
    ptrdiff_t *info
);

/* Source: dlaeda.f */
#define dlaeda FORTRAN_WRAPPER(dlaeda)
extern void dlaeda(
    ptrdiff_t *n,
    ptrdiff_t *tlvls,
    ptrdiff_t *curlvl,
    ptrdiff_t *curpbm,
    ptrdiff_t *prmptr,
    ptrdiff_t *perm,
    ptrdiff_t *givptr,
    ptrdiff_t *givcol,
    double *givnum,
    double *q,
    ptrdiff_t *qptr,
    double *z,
    double *ztemp,
    ptrdiff_t *info
);

/* Source: dlaein.f */
#define dlaein FORTRAN_WRAPPER(dlaein)
extern void dlaein(
    ptrdiff_t *rightv,
    ptrdiff_t *noinit,
    ptrdiff_t *n,
    double *h,
    ptrdiff_t *ldh,
    double *wr,
    double *wi,
    double *vr,
    double *vi,
    double *b,
    ptrdiff_t *ldb,
    double *work,
    double *eps3,
    double *smlnum,
    double *bignum,
    ptrdiff_t *info
);

/* Source: dlaev2.f */
#define dlaev2 FORTRAN_WRAPPER(dlaev2)
extern void dlaev2(
    double *a,
    double *b,
    double *c,
    double *rt1,
    double *rt2,
    double *cs1,
    double *sn1
);

/* Source: dlaexc.f */
#define dlaexc FORTRAN_WRAPPER(dlaexc)
extern void dlaexc(
    ptrdiff_t *wantq,
    ptrdiff_t *n,
    double *t,
    ptrdiff_t *ldt,
    double *q,
    ptrdiff_t *ldq,
    ptrdiff_t *j1_,
    ptrdiff_t *n1,
    ptrdiff_t *n2,
    double *work,
    ptrdiff_t *info
);

/* Source: dlag2.f */
#define dlag2 FORTRAN_WRAPPER(dlag2)
extern void dlag2(
    double *a,
    ptrdiff_t *lda,
    double *b,
    ptrdiff_t *ldb,
    double *safmin,
    double *scale1,
    double *scale2,
    double *wr1,
    double *wr2,
    double *wi
);

/* Source: dlag2s.f */
#define dlag2s FORTRAN_WRAPPER(dlag2s)
extern void dlag2s(
    ptrdiff_t *m,
    ptrdiff_t *n,
    double *a,
    ptrdiff_t *lda,
    float  *sa,
    ptrdiff_t *ldsa,
    ptrdiff_t *info
);

/* Source: dlags2.f */
#define dlags2 FORTRAN_WRAPPER(dlags2)
extern void dlags2(
    ptrdiff_t *upper,
    double *a1,
    double *a2,
    double *a3,
    double *b1,
    double *b2,
    double *b3,
    double *csu,
    double *snu,
    double *csv,
    double *snv,
    double *csq,
    double *snq
);

/* Source: dlagtf.f */
#define dlagtf FORTRAN_WRAPPER(dlagtf)
extern void dlagtf(
    ptrdiff_t *n,
    double *a,
    double *lambda,
    double *b,
    double *c,
    double *tol,
    double *d,
    ptrdiff_t *in,
    ptrdiff_t *info
);

/* Source: dlagtm.f */
#define dlagtm FORTRAN_WRAPPER(dlagtm)
extern void dlagtm(
    char   *trans,
    ptrdiff_t *n,
    ptrdiff_t *nrhs,
    double *alpha,
    double *dl,
    double *d,
    double *du,
    double *x,
    ptrdiff_t *ldx,
    double *beta,
    double *b,
    ptrdiff_t *ldb
);

/* Source: dlagts.f */
#define dlagts FORTRAN_WRAPPER(dlagts)
extern void dlagts(
    ptrdiff_t *job,
    ptrdiff_t *n,
    double *a,
    double *b,
    double *c,
    double *d,
    ptrdiff_t *in,
    double *y,
    double *tol,
    ptrdiff_t *info
);

/* Source: dlagv2.f */
#define dlagv2 FORTRAN_WRAPPER(dlagv2)
extern void dlagv2(
    double *a,
    ptrdiff_t *lda,
    double *b,
    ptrdiff_t *ldb,
    double *alphar,
    double *alphai,
    double *beta,
    double *csl,
    double *snl,
    double *csr,
    double *snr
);

/* Source: dlahqr.f */
#define dlahqr FORTRAN_WRAPPER(dlahqr)
extern void dlahqr(
    ptrdiff_t *wantt,
    ptrdiff_t *wantz,
    ptrdiff_t *n,
    ptrdiff_t *ilo,
    ptrdiff_t *ihi,
    double *h,
    ptrdiff_t *ldh,
    double *wr,
    double *wi,
    ptrdiff_t *iloz,
    ptrdiff_t *ihiz,
    double *z,
    ptrdiff_t *ldz,
    ptrdiff_t *info
);

/* Source: dlahr2.f */
#define dlahr2 FORTRAN_WRAPPER(dlahr2)
extern void dlahr2(
    ptrdiff_t *n,
    ptrdiff_t *k,
    ptrdiff_t *nb,
    double *a,
    ptrdiff_t *lda,
    double *tau,
    double *t,
    ptrdiff_t *ldt,
    double *y,
    ptrdiff_t *ldy
);

/* Source: dlahrd.f */
#define dlahrd FORTRAN_WRAPPER(dlahrd)
extern void dlahrd(
    ptrdiff_t *n,
    ptrdiff_t *k,
    ptrdiff_t *nb,
    double *a,
    ptrdiff_t *lda,
    double *tau,
    double *t,
    ptrdiff_t *ldt,
    double *y,
    ptrdiff_t *ldy
);

/* Source: dlaic1.f */
#define dlaic1 FORTRAN_WRAPPER(dlaic1)
extern void dlaic1(
    ptrdiff_t *job,
    ptrdiff_t *j,
    double *x,
    double *sest,
    double *w,
    double *gamma_,
    double *sestpr,
    double *s,
    double *c
);

/* Source: dlaisnan.f */
#define dlaisnan FORTRAN_WRAPPER(dlaisnan)
extern ptrdiff_t dlaisnan(
    double *din1,
    double *din2
);

/* Source: dlaln2.f */
#define dlaln2 FORTRAN_WRAPPER(dlaln2)
extern void dlaln2(
    ptrdiff_t *ltrans,
    ptrdiff_t *na,
    ptrdiff_t *nw,
    double *smin,
    double *ca,
    double *a,
    ptrdiff_t *lda,
    double *d1,
    double *d2,
    double *b,
    ptrdiff_t *ldb,
    double *wr,
    double *wi,
    double *x,
    ptrdiff_t *ldx,
    double *scale,
    double *xnorm,
    ptrdiff_t *info
);

/* Source: dlals0.f */
#define dlals0 FORTRAN_WRAPPER(dlals0)
extern void dlals0(
    ptrdiff_t *icompq,
    ptrdiff_t *nl,
    ptrdiff_t *nr,
    ptrdiff_t *sqre,
    ptrdiff_t *nrhs,
    double *b,
    ptrdiff_t *ldb,
    double *bx,
    ptrdiff_t *ldbx,
    ptrdiff_t *perm,
    ptrdiff_t *givptr,
    ptrdiff_t *givcol,
    ptrdiff_t *ldgcol,
    double *givnum,
    ptrdiff_t *ldgnum,
    double *poles,
    double *difl,
    double *difr,
    double *z,
    ptrdiff_t *k,
    double *c,
    double *s,
    double *work,
    ptrdiff_t *info
);

/* Source: dlalsa.f */
#define dlalsa FORTRAN_WRAPPER(dlalsa)
extern void dlalsa(
    ptrdiff_t *icompq,
    ptrdiff_t *smlsiz,
    ptrdiff_t *n,
    ptrdiff_t *nrhs,
    double *b,
    ptrdiff_t *ldb,
    double *bx,
    ptrdiff_t *ldbx,
    double *u,
    ptrdiff_t *ldu,
    double *vt,
    ptrdiff_t *k,
    double *difl,
    double *difr,
    double *z,
    double *poles,
    ptrdiff_t *givptr,
    ptrdiff_t *givcol,
    ptrdiff_t *ldgcol,
    ptrdiff_t *perm,
    double *givnum,
    double *c,
    double *s,
    double *work,
    ptrdiff_t *iwork,
    ptrdiff_t *info
);

/* Source: dlalsd.f */
#define dlalsd FORTRAN_WRAPPER(dlalsd)
extern void dlalsd(
    char   *uplo,
    ptrdiff_t *smlsiz,
    ptrdiff_t *n,
    ptrdiff_t *nrhs,
    double *d,
    double *e,
    double *b,
    ptrdiff_t *ldb,
    double *rcond,
    ptrdiff_t *rank,
    double *work,
    ptrdiff_t *iwork,
    ptrdiff_t *info
);

/* Source: dlamrg.f */
#define dlamrg FORTRAN_WRAPPER(dlamrg)
extern void dlamrg(
    ptrdiff_t *n1,
    ptrdiff_t *n2,
    double *a,
    ptrdiff_t *dtrd1,
    ptrdiff_t *dtrd2,
    ptrdiff_t *index
);

/* Source: dlaneg.f */
#define dlaneg FORTRAN_WRAPPER(dlaneg)
extern ptrdiff_t dlaneg(
    ptrdiff_t *n,
    double *d,
    double *lld,
    double *sigma,
    double *pivmin,
    ptrdiff_t *r
);

/* Source: dlangb.f */
#define dlangb FORTRAN_WRAPPER(dlangb)
extern double dlangb(
    char   *norm,
    ptrdiff_t *n,
    ptrdiff_t *kl,
    ptrdiff_t *ku,
    double *ab,
    ptrdiff_t *ldab,
    double *work
);

/* Source: dlange.f */
#define dlange FORTRAN_WRAPPER(dlange)
extern double dlange(
    char   *norm,
    ptrdiff_t *m,
    ptrdiff_t *n,
    double *a,
    ptrdiff_t *lda,
    double *work
);

/* Source: dlangt.f */
#define dlangt FORTRAN_WRAPPER(dlangt)
extern double dlangt(
    char   *norm,
    ptrdiff_t *n,
    double *dl,
    double *d,
    double *du
);

/* Source: dlanhs.f */
#define dlanhs FORTRAN_WRAPPER(dlanhs)
extern double dlanhs(
    char   *norm,
    ptrdiff_t *n,
    double *a,
    ptrdiff_t *lda,
    double *work
);

/* Source: dlansb.f */
#define dlansb FORTRAN_WRAPPER(dlansb)
extern double dlansb(
    char   *norm,
    char   *uplo,
    ptrdiff_t *n,
    ptrdiff_t *k,
    double *ab,
    ptrdiff_t *ldab,
    double *work
);

/* Source: dlansf.f */
#define dlansf FORTRAN_WRAPPER(dlansf)
extern double dlansf(
    char   *norm,
    char   *transr,
    char   *uplo,
    ptrdiff_t *n,
    double *a,
    double *work
);

/* Source: dlansp.f */
#define dlansp FORTRAN_WRAPPER(dlansp)
extern double dlansp(
    char   *norm,
    char   *uplo,
    ptrdiff_t *n,
    double *ap,
    double *work
);

/* Source: dlanst.f */
#define dlanst FORTRAN_WRAPPER(dlanst)
extern double dlanst(
    char   *norm,
    ptrdiff_t *n,
    double *d,
    double *e
);

/* Source: dlansy.f */
#define dlansy FORTRAN_WRAPPER(dlansy)
extern double dlansy(
    char   *norm,
    char   *uplo,
    ptrdiff_t *n,
    double *a,
    ptrdiff_t *lda,
    double *work
);

/* Source: dlantb.f */
#define dlantb FORTRAN_WRAPPER(dlantb)
extern double dlantb(
    char   *norm,
    char   *uplo,
    char   *diag,
    ptrdiff_t *n,
    ptrdiff_t *k,
    double *ab,
    ptrdiff_t *ldab,
    double *work
);

/* Source: dlantp.f */
#define dlantp FORTRAN_WRAPPER(dlantp)
extern double dlantp(
    char   *norm,
    char   *uplo,
    char   *diag,
    ptrdiff_t *n,
    double *ap,
    double *work
);

/* Source: dlantr.f */
#define dlantr FORTRAN_WRAPPER(dlantr)
extern double dlantr(
    char   *norm,
    char   *uplo,
    char   *diag,
    ptrdiff_t *m,
    ptrdiff_t *n,
    double *a,
    ptrdiff_t *lda,
    double *work
);

/* Source: dlanv2.f */
#define dlanv2 FORTRAN_WRAPPER(dlanv2)
extern void dlanv2(
    double *a,
    double *b,
    double *c,
    double *d,
    double *rt1r,
    double *rt1i,
    double *rt2r,
    double *rt2i,
    double *cs,
    double *sn
);

/* Source: dlapll.f */
#define dlapll FORTRAN_WRAPPER(dlapll)
extern void dlapll(
    ptrdiff_t *n,
    double *x,
    ptrdiff_t *incx,
    double *y,
    ptrdiff_t *incy,
    double *ssmin
);

/* Source: dlapmt.f */
#define dlapmt FORTRAN_WRAPPER(dlapmt)
extern void dlapmt(
    ptrdiff_t *forwrd,
    ptrdiff_t *m,
    ptrdiff_t *n,
    double *x,
    ptrdiff_t *ldx,
    ptrdiff_t *k
);

/* Source: dlapy2.f */
#define dlapy2 FORTRAN_WRAPPER(dlapy2)
extern double dlapy2(
    double *x,
    double *y
);

/* Source: dlapy3.f */
#define dlapy3 FORTRAN_WRAPPER(dlapy3)
extern double dlapy3(
    double *x,
    double *y,
    double *z
);

/* Source: dlaqgb.f */
#define dlaqgb FORTRAN_WRAPPER(dlaqgb)
extern void dlaqgb(
    ptrdiff_t *m,
    ptrdiff_t *n,
    ptrdiff_t *kl,
    ptrdiff_t *ku,
    double *ab,
    ptrdiff_t *ldab,
    double *r,
    double *c,
    double *rowcnd,
    double *colcnd,
    double *amax,
    char   *equed
);

/* Source: dlaqge.f */
#define dlaqge FORTRAN_WRAPPER(dlaqge)
extern void dlaqge(
    ptrdiff_t *m,
    ptrdiff_t *n,
    double *a,
    ptrdiff_t *lda,
    double *r,
    double *c,
    double *rowcnd,
    double *colcnd,
    double *amax,
    char   *equed
);

/* Source: dlaqp2.f */
#define dlaqp2 FORTRAN_WRAPPER(dlaqp2)
extern void dlaqp2(
    ptrdiff_t *m,
    ptrdiff_t *n,
    ptrdiff_t *offset,
    double *a,
    ptrdiff_t *lda,
    ptrdiff_t *jpvt,
    double *tau,
    double *vn1,
    double *vn2,
    double *work
);

/* Source: dlaqps.f */
#define dlaqps FORTRAN_WRAPPER(dlaqps)
extern void dlaqps(
    ptrdiff_t *m,
    ptrdiff_t *n,
    ptrdiff_t *offset,
    ptrdiff_t *nb,
    ptrdiff_t *kb,
    double *a,
    ptrdiff_t *lda,
    ptrdiff_t *jpvt,
    double *tau,
    double *vn1,
    double *vn2,
    double *auxv,
    double *f,
    ptrdiff_t *ldf
);

/* Source: dlaqr0.f */
#define dlaqr0 FORTRAN_WRAPPER(dlaqr0)
extern void dlaqr0(
    ptrdiff_t *wantt,
    ptrdiff_t *wantz,
    ptrdiff_t *n,
    ptrdiff_t *ilo,
    ptrdiff_t *ihi,
    double *h,
    ptrdiff_t *ldh,
    double *wr,
    double *wi,
    ptrdiff_t *iloz,
    ptrdiff_t *ihiz,
    double *z,
    ptrdiff_t *ldz,
    double *work,
    ptrdiff_t *lwork,
    ptrdiff_t *info
);

/* Source: dlaqr1.f */
#define dlaqr1 FORTRAN_WRAPPER(dlaqr1)
extern void dlaqr1(
    ptrdiff_t *n,
    double *h,
    ptrdiff_t *ldh,
    double *sr1,
    double *si1,
    double *sr2,
    double *si2,
    double *v
);

/* Source: dlaqr2.f */
#define dlaqr2 FORTRAN_WRAPPER(dlaqr2)
extern void dlaqr2(
    ptrdiff_t *wantt,
    ptrdiff_t *wantz,
    ptrdiff_t *n,
    ptrdiff_t *ktop,
    ptrdiff_t *kbot,
    ptrdiff_t *nw,
    double *h,
    ptrdiff_t *ldh,
    ptrdiff_t *iloz,
    ptrdiff_t *ihiz,
    double *z,
    ptrdiff_t *ldz,
    ptrdiff_t *ns,
    ptrdiff_t *nd,
    double *sr,
    double *si,
    double *v,
    ptrdiff_t *ldv,
    ptrdiff_t *nh,
    double *t,
    ptrdiff_t *ldt,
    ptrdiff_t *nv,
    double *wv,
    ptrdiff_t *ldwv,
    double *work,
    ptrdiff_t *lwork
);

/* Source: dlaqr3.f */
#define dlaqr3 FORTRAN_WRAPPER(dlaqr3)
extern void dlaqr3(
    ptrdiff_t *wantt,
    ptrdiff_t *wantz,
    ptrdiff_t *n,
    ptrdiff_t *ktop,
    ptrdiff_t *kbot,
    ptrdiff_t *nw,
    double *h,
    ptrdiff_t *ldh,
    ptrdiff_t *iloz,
    ptrdiff_t *ihiz,
    double *z,
    ptrdiff_t *ldz,
    ptrdiff_t *ns,
    ptrdiff_t *nd,
    double *sr,
    double *si,
    double *v,
    ptrdiff_t *ldv,
    ptrdiff_t *nh,
    double *t,
    ptrdiff_t *ldt,
    ptrdiff_t *nv,
    double *wv,
    ptrdiff_t *ldwv,
    double *work,
    ptrdiff_t *lwork
);

/* Source: dlaqr4.f */
#define dlaqr4 FORTRAN_WRAPPER(dlaqr4)
extern void dlaqr4(
    ptrdiff_t *wantt,
    ptrdiff_t *wantz,
    ptrdiff_t *n,
    ptrdiff_t *ilo,
    ptrdiff_t *ihi,
    double *h,
    ptrdiff_t *ldh,
    double *wr,
    double *wi,
    ptrdiff_t *iloz,
    ptrdiff_t *ihiz,
    double *z,
    ptrdiff_t *ldz,
    double *work,
    ptrdiff_t *lwork,
    ptrdiff_t *info
);

/* Source: dlaqr5.f */
#define dlaqr5 FORTRAN_WRAPPER(dlaqr5)
extern void dlaqr5(
    ptrdiff_t *wantt,
    ptrdiff_t *wantz,
    ptrdiff_t *kacc22,
    ptrdiff_t *n,
    ptrdiff_t *ktop,
    ptrdiff_t *kbot,
    ptrdiff_t *nshfts,
    double *sr,
    double *si,
    double *h,
    ptrdiff_t *ldh,
    ptrdiff_t *iloz,
    ptrdiff_t *ihiz,
    double *z,
    ptrdiff_t *ldz,
    double *v,
    ptrdiff_t *ldv,
    double *u,
    ptrdiff_t *ldu,
    ptrdiff_t *nv,
    double *wv,
    ptrdiff_t *ldwv,
    ptrdiff_t *nh,
    double *wh,
    ptrdiff_t *ldwh
);

/* Source: dlaqsb.f */
#define dlaqsb FORTRAN_WRAPPER(dlaqsb)
extern void dlaqsb(
    char   *uplo,
    ptrdiff_t *n,
    ptrdiff_t *kd,
    double *ab,
    ptrdiff_t *ldab,
    double *s,
    double *scond,
    double *amax,
    char   *equed
);

/* Source: dlaqsp.f */
#define dlaqsp FORTRAN_WRAPPER(dlaqsp)
extern void dlaqsp(
    char   *uplo,
    ptrdiff_t *n,
    double *ap,
    double *s,
    double *scond,
    double *amax,
    char   *equed
);

/* Source: dlaqsy.f */
#define dlaqsy FORTRAN_WRAPPER(dlaqsy)
extern void dlaqsy(
    char   *uplo,
    ptrdiff_t *n,
    double *a,
    ptrdiff_t *lda,
    double *s,
    double *scond,
    double *amax,
    char   *equed
);

/* Source: dlaqtr.f */
#define dlaqtr FORTRAN_WRAPPER(dlaqtr)
extern void dlaqtr(
    ptrdiff_t *ltran,
    ptrdiff_t *lreal,
    ptrdiff_t *n,
    double *t,
    ptrdiff_t *ldt,
    double *b,
    double *w,
    double *scale,
    double *x,
    double *work,
    ptrdiff_t *info
);

/* Source: dlar1v.f */
#define dlar1v FORTRAN_WRAPPER(dlar1v)
extern void dlar1v(
    ptrdiff_t *n,
    ptrdiff_t *b1,
    ptrdiff_t *bn,
    double *lambda,
    double *d,
    double *l,
    double *ld,
    double *lld,
    double *pivmin,
    double *gaptol,
    double *z,
    ptrdiff_t *wantnc,
    ptrdiff_t *negcnt,
    double *ztz,
    double *mingma,
    ptrdiff_t *r,
    ptrdiff_t *isuppz,
    double *nrminv,
    double *resid,
    double *rqcorr,
    double *work
);

/* Source: dlar2v.f */
#define dlar2v FORTRAN_WRAPPER(dlar2v)
extern void dlar2v(
    ptrdiff_t *n,
    double *x,
    double *y,
    double *z,
    ptrdiff_t *incx,
    double *c,
    double *s,
    ptrdiff_t *incc
);

/* Source: dlarf.f */
#define dlarf FORTRAN_WRAPPER(dlarf)
extern void dlarf(
    char   *side,
    ptrdiff_t *m,
    ptrdiff_t *n,
    double *v,
    ptrdiff_t *incv,
    double *tau,
    double *c,
    ptrdiff_t *ldc,
    double *work
);

/* Source: dlarfb.f */
#define dlarfb FORTRAN_WRAPPER(dlarfb)
extern void dlarfb(
    char   *side,
    char   *trans,
    char   *direct,
    char   *storev,
    ptrdiff_t *m,
    ptrdiff_t *n,
    ptrdiff_t *k,
    double *v,
    ptrdiff_t *ldv,
    double *t,
    ptrdiff_t *ldt,
    double *c,
    ptrdiff_t *ldc,
    double *work,
    ptrdiff_t *ldwork
);

/* Source: dlarfg.f */
#define dlarfg FORTRAN_WRAPPER(dlarfg)
extern void dlarfg(
    ptrdiff_t *n,
    double *alpha,
    double *x,
    ptrdiff_t *incx,
    double *tau
);

/* Source: dlarfgp.f */
#define dlarfgp FORTRAN_WRAPPER(dlarfgp)
extern void dlarfgp(
    ptrdiff_t *n,
    double *alpha,
    double *x,
    ptrdiff_t *incx,
    double *tau
);

/* Source: dlarft.f */
#define dlarft FORTRAN_WRAPPER(dlarft)
extern void dlarft(
    char   *direct,
    char   *storev,
    ptrdiff_t *n,
    ptrdiff_t *k,
    double *v,
    ptrdiff_t *ldv,
    double *tau,
    double *t,
    ptrdiff_t *ldt
);

/* Source: dlarfx.f */
#define dlarfx FORTRAN_WRAPPER(dlarfx)
extern void dlarfx(
    char   *side,
    ptrdiff_t *m,
    ptrdiff_t *n,
    double *v,
    double *tau,
    double *c,
    ptrdiff_t *ldc,
    double *work
);

/* Source: dlargv.f */
#define dlargv FORTRAN_WRAPPER(dlargv)
extern void dlargv(
    ptrdiff_t *n,
    double *x,
    ptrdiff_t *incx,
    double *y,
    ptrdiff_t *incy,
    double *c,
    ptrdiff_t *incc
);

/* Source: dlarnv.f */
#define dlarnv FORTRAN_WRAPPER(dlarnv)
extern void dlarnv(
    ptrdiff_t *idist,
    ptrdiff_t *iseed,
    ptrdiff_t *n,
    double *x
);

/* Source: dlarra.f */
#define dlarra FORTRAN_WRAPPER(dlarra)
extern void dlarra(
    ptrdiff_t *n,
    double *d,
    double *e,
    double *e2,
    double *spltol,
    double *tnrm,
    ptrdiff_t *nsplit,
    ptrdiff_t *isplit,
    ptrdiff_t *info
);

/* Source: dlarrb.f */
#define dlarrb FORTRAN_WRAPPER(dlarrb)
extern void dlarrb(
    ptrdiff_t *n,
    double *d,
    double *lld,
    ptrdiff_t *ifirst,
    ptrdiff_t *ilast,
    double *rtol1,
    double *rtol2,
    ptrdiff_t *offset,
    double *w,
    double *wgap,
    double *werr,
    double *work,
    ptrdiff_t *iwork,
    double *pivmin,
    double *spdiam,
    ptrdiff_t *twist,
    ptrdiff_t *info
);

/* Source: dlarrc.f */
#define dlarrc FORTRAN_WRAPPER(dlarrc)
extern void dlarrc(
    char   *jobt,
    ptrdiff_t *n,
    double *vl,
    double *vu,
    double *d,
    double *e,
    double *pivmin,
    ptrdiff_t *eigcnt,
    ptrdiff_t *lcnt,
    ptrdiff_t *rcnt,
    ptrdiff_t *info
);

/* Source: dlarrd.f */
#define dlarrd FORTRAN_WRAPPER(dlarrd)
extern void dlarrd(
    char   *range,
    char   *order,
    ptrdiff_t *n,
    double *vl,
    double *vu,
    ptrdiff_t *il,
    ptrdiff_t *iu,
    double *gers,
    double *reltol,
    double *d,
    double *e,
    double *e2,
    double *pivmin,
    ptrdiff_t *nsplit,
    ptrdiff_t *isplit,
    ptrdiff_t *m,
    double *w,
    double *werr,
    double *wl,
    double *wu,
    ptrdiff_t *iblock,
    ptrdiff_t *indexw,
    double *work,
    ptrdiff_t *iwork,
    ptrdiff_t *info
);

/* Source: dlarre.f */
#define dlarre FORTRAN_WRAPPER(dlarre)
extern void dlarre(
    char   *range,
    ptrdiff_t *n,
    double *vl,
    double *vu,
    ptrdiff_t *il,
    ptrdiff_t *iu,
    double *d,
    double *e,
    double *e2,
    double *rtol1,
    double *rtol2,
    double *spltol,
    ptrdiff_t *nsplit,
    ptrdiff_t *isplit,
    ptrdiff_t *m,
    double *w,
    double *werr,
    double *wgap,
    ptrdiff_t *iblock,
    ptrdiff_t *indexw,
    double *gers,
    double *pivmin,
    double *work,
    ptrdiff_t *iwork,
    ptrdiff_t *info
);

/* Source: dlarrf.f */
#define dlarrf FORTRAN_WRAPPER(dlarrf)
extern void dlarrf(
    ptrdiff_t *n,
    double *d,
    double *l,
    double *ld,
    ptrdiff_t *clstrt,
    ptrdiff_t *clend,
    double *w,
    double *wgap,
    double *werr,
    double *spdiam,
    double *clgapl,
    double *clgapr,
    double *pivmin,
    double *sigma,
    double *dplus,
    double *lplus,
    double *work,
    ptrdiff_t *info
);

/* Source: dlarrj.f */
#define dlarrj FORTRAN_WRAPPER(dlarrj)
extern void dlarrj(
    ptrdiff_t *n,
    double *d,
    double *e2,
    ptrdiff_t *ifirst,
    ptrdiff_t *ilast,
    double *rtol,
    ptrdiff_t *offset,
    double *w,
    double *werr,
    double *work,
    ptrdiff_t *iwork,
    double *pivmin,
    double *spdiam,
    ptrdiff_t *info
);

/* Source: dlarrk.f */
#define dlarrk FORTRAN_WRAPPER(dlarrk)
extern void dlarrk(
    ptrdiff_t *n,
    ptrdiff_t *iw,
    double *gl,
    double *gu,
    double *d,
    double *e2,
    double *pivmin,
    double *reltol,
    double *w,
    double *werr,
    ptrdiff_t *info
);

/* Source: dlarrr.f */
#define dlarrr FORTRAN_WRAPPER(dlarrr)
extern void dlarrr(
    ptrdiff_t *n,
    double *d,
    double *e,
    ptrdiff_t *info
);

/* Source: dlarrv.f */
#define dlarrv FORTRAN_WRAPPER(dlarrv)
extern void dlarrv(
    ptrdiff_t *n,
    double *vl,
    double *vu,
    double *d,
    double *l,
    double *pivmin,
    ptrdiff_t *isplit,
    ptrdiff_t *m,
    ptrdiff_t *dol,
    ptrdiff_t *dou,
    double *minrgp,
    double *rtol1,
    double *rtol2,
    double *w,
    double *werr,
    double *wgap,
    ptrdiff_t *iblock,
    ptrdiff_t *indexw,
    double *gers,
    double *z,
    ptrdiff_t *ldz,
    ptrdiff_t *isuppz,
    double *work,
    ptrdiff_t *iwork,
    ptrdiff_t *info
);

/* Source: dlartg.f */
#define dlartg FORTRAN_WRAPPER(dlartg)
extern void dlartg(
    double *f,
    double *g,
    double *cs,
    double *sn,
    double *r
);

/* Source: dlartv.f */
#define dlartv FORTRAN_WRAPPER(dlartv)
extern void dlartv(
    ptrdiff_t *n,
    double *x,
    ptrdiff_t *incx,
    double *y,
    ptrdiff_t *incy,
    double *c,
    double *s,
    ptrdiff_t *incc
);

/* Source: dlaruv.f */
#define dlaruv FORTRAN_WRAPPER(dlaruv)
extern void dlaruv(
    ptrdiff_t *iseed,
    ptrdiff_t *n,
    double *x
);

/* Source: dlarz.f */
#define dlarz FORTRAN_WRAPPER(dlarz)
extern void dlarz(
    char   *side,
    ptrdiff_t *m,
    ptrdiff_t *n,
    ptrdiff_t *l,
    double *v,
    ptrdiff_t *incv,
    double *tau,
    double *c,
    ptrdiff_t *ldc,
    double *work
);

/* Source: dlarzb.f */
#define dlarzb FORTRAN_WRAPPER(dlarzb)
extern void dlarzb(
    char   *side,
    char   *trans,
    char   *direct,
    char   *storev,
    ptrdiff_t *m,
    ptrdiff_t *n,
    ptrdiff_t *k,
    ptrdiff_t *l,
    double *v,
    ptrdiff_t *ldv,
    double *t,
    ptrdiff_t *ldt,
    double *c,
    ptrdiff_t *ldc,
    double *work,
    ptrdiff_t *ldwork
);

/* Source: dlarzt.f */
#define dlarzt FORTRAN_WRAPPER(dlarzt)
extern void dlarzt(
    char   *direct,
    char   *storev,
    ptrdiff_t *n,
    ptrdiff_t *k,
    double *v,
    ptrdiff_t *ldv,
    double *tau,
    double *t,
    ptrdiff_t *ldt
);

/* Source: dlas2.f */
#define dlas2 FORTRAN_WRAPPER(dlas2)
extern void dlas2(
    double *f,
    double *g,
    double *h,
    double *ssmin,
    double *ssmax
);

/* Source: dlascl.f */
#define dlascl FORTRAN_WRAPPER(dlascl)
extern void dlascl(
    char   *type,
    ptrdiff_t *kl,
    ptrdiff_t *ku,
    double *cfrom,
    double *cto,
    ptrdiff_t *m,
    ptrdiff_t *n,
    double *a,
    ptrdiff_t *lda,
    ptrdiff_t *info
);

/* Source: dlasd0.f */
#define dlasd0 FORTRAN_WRAPPER(dlasd0)
extern void dlasd0(
    ptrdiff_t *n,
    ptrdiff_t *sqre,
    double *d,
    double *e,
    double *u,
    ptrdiff_t *ldu,
    double *vt,
    ptrdiff_t *ldvt,
    ptrdiff_t *smlsiz,
    ptrdiff_t *iwork,
    double *work,
    ptrdiff_t *info
);

/* Source: dlasd1.f */
#define dlasd1 FORTRAN_WRAPPER(dlasd1)
extern void dlasd1(
    ptrdiff_t *nl,
    ptrdiff_t *nr,
    ptrdiff_t *sqre,
    double *d,
    double *alpha,
    double *beta,
    double *u,
    ptrdiff_t *ldu,
    double *vt,
    ptrdiff_t *ldvt,
    ptrdiff_t *idxq,
    ptrdiff_t *iwork,
    double *work,
    ptrdiff_t *info
);

/* Source: dlasd2.f */
#define dlasd2 FORTRAN_WRAPPER(dlasd2)
extern void dlasd2(
    ptrdiff_t *nl,
    ptrdiff_t *nr,
    ptrdiff_t *sqre,
    ptrdiff_t *k,
    double *d,
    double *z,
    double *alpha,
    double *beta,
    double *u,
    ptrdiff_t *ldu,
    double *vt,
    ptrdiff_t *ldvt,
    double *dsigma,
    double *u2,
    ptrdiff_t *ldu2,
    double *vt2,
    ptrdiff_t *ldvt2,
    ptrdiff_t *idxp,
    ptrdiff_t *idx,
    ptrdiff_t *idxc,
    ptrdiff_t *idxq,
    ptrdiff_t *coltyp,
    ptrdiff_t *info
);

/* Source: dlasd3.f */
#define dlasd3 FORTRAN_WRAPPER(dlasd3)
extern void dlasd3(
    ptrdiff_t *nl,
    ptrdiff_t *nr,
    ptrdiff_t *sqre,
    ptrdiff_t *k,
    double *d,
    double *q,
    ptrdiff_t *ldq,
    double *dsigma,
    double *u,
    ptrdiff_t *ldu,
    double *u2,
    ptrdiff_t *ldu2,
    double *vt,
    ptrdiff_t *ldvt,
    double *vt2,
    ptrdiff_t *ldvt2,
    ptrdiff_t *idxc,
    ptrdiff_t *ctot,
    double *z,
    ptrdiff_t *info
);

/* Source: dlasd4.f */
#define dlasd4 FORTRAN_WRAPPER(dlasd4)
extern void dlasd4(
    ptrdiff_t *n,
    ptrdiff_t *i,
    double *d,
    double *z,
    double *delta,
    double *rho,
    double *sigma,
    double *work,
    ptrdiff_t *info
);

/* Source: dlasd5.f */
#define dlasd5 FORTRAN_WRAPPER(dlasd5)
extern void dlasd5(
    ptrdiff_t *i,
    double *d,
    double *z,
    double *delta,
    double *rho,
    double *dsigma,
    double *work
);

/* Source: dlasd6.f */
#define dlasd6 FORTRAN_WRAPPER(dlasd6)
extern void dlasd6(
    ptrdiff_t *icompq,
    ptrdiff_t *nl,
    ptrdiff_t *nr,
    ptrdiff_t *sqre,
    double *d,
    double *vf,
    double *vl,
    double *alpha,
    double *beta,
    ptrdiff_t *idxq,
    ptrdiff_t *perm,
    ptrdiff_t *givptr,
    ptrdiff_t *givcol,
    ptrdiff_t *ldgcol,
    double *givnum,
    ptrdiff_t *ldgnum,
    double *poles,
    double *difl,
    double *difr,
    double *z,
    ptrdiff_t *k,
    double *c,
    double *s,
    double *work,
    ptrdiff_t *iwork,
    ptrdiff_t *info
);

/* Source: dlasd7.f */
#define dlasd7 FORTRAN_WRAPPER(dlasd7)
extern void dlasd7(
    ptrdiff_t *icompq,
    ptrdiff_t *nl,
    ptrdiff_t *nr,
    ptrdiff_t *sqre,
    ptrdiff_t *k,
    double *d,
    double *z,
    double *zw,
    double *vf,
    double *vfw,
    double *vl,
    double *vlw,
    double *alpha,
    double *beta,
    double *dsigma,
    ptrdiff_t *idx,
    ptrdiff_t *idxp,
    ptrdiff_t *idxq,
    ptrdiff_t *perm,
    ptrdiff_t *givptr,
    ptrdiff_t *givcol,
    ptrdiff_t *ldgcol,
    double *givnum,
    ptrdiff_t *ldgnum,
    double *c,
    double *s,
    ptrdiff_t *info
);

/* Source: dlasd8.f */
#define dlasd8 FORTRAN_WRAPPER(dlasd8)
extern void dlasd8(
    ptrdiff_t *icompq,
    ptrdiff_t *k,
    double *d,
    double *z,
    double *vf,
    double *vl,
    double *difl,
    double *difr,
    ptrdiff_t *lddifr,
    double *dsigma,
    double *work,
    ptrdiff_t *info
);

/* Source: dlasda.f */
#define dlasda FORTRAN_WRAPPER(dlasda)
extern void dlasda(
    ptrdiff_t *icompq,
    ptrdiff_t *smlsiz,
    ptrdiff_t *n,
    ptrdiff_t *sqre,
    double *d,
    double *e,
    double *u,
    ptrdiff_t *ldu,
    double *vt,
    ptrdiff_t *k,
    double *difl,
    double *difr,
    double *z,
    double *poles,
    ptrdiff_t *givptr,
    ptrdiff_t *givcol,
    ptrdiff_t *ldgcol,
    ptrdiff_t *perm,
    double *givnum,
    double *c,
    double *s,
    double *work,
    ptrdiff_t *iwork,
    ptrdiff_t *info
);

/* Source: dlasdq.f */
#define dlasdq FORTRAN_WRAPPER(dlasdq)
extern void dlasdq(
    char   *uplo,
    ptrdiff_t *sqre,
    ptrdiff_t *n,
    ptrdiff_t *ncvt,
    ptrdiff_t *nru,
    ptrdiff_t *ncc,
    double *d,
    double *e,
    double *vt,
    ptrdiff_t *ldvt,
    double *u,
    ptrdiff_t *ldu,
    double *c,
    ptrdiff_t *ldc,
    double *work,
    ptrdiff_t *info
);

/* Source: dlasdt.f */
#define dlasdt FORTRAN_WRAPPER(dlasdt)
extern void dlasdt(
    ptrdiff_t *n,
    ptrdiff_t *lvl,
    ptrdiff_t *nd,
    ptrdiff_t *inode,
    ptrdiff_t *ndiml,
    ptrdiff_t *ndimr,
    ptrdiff_t *msub
);

/* Source: dlaset.f */
#define dlaset FORTRAN_WRAPPER(dlaset)
extern void dlaset(
    char   *uplo,
    ptrdiff_t *m,
    ptrdiff_t *n,
    double *alpha,
    double *beta,
    double *a,
    ptrdiff_t *lda
);

/* Source: dlasq1.f */
#define dlasq1 FORTRAN_WRAPPER(dlasq1)
extern void dlasq1(
    ptrdiff_t *n,
    double *d,
    double *e,
    double *work,
    ptrdiff_t *info
);

/* Source: dlasq2.f */
#define dlasq2 FORTRAN_WRAPPER(dlasq2)
extern void dlasq2(
    ptrdiff_t *n,
    double *z,
    ptrdiff_t *info
);

/* Source: dlasq3.f */
#define dlasq3 FORTRAN_WRAPPER(dlasq3)
extern void dlasq3(
    ptrdiff_t *i0,
    ptrdiff_t *n0,
    double *z,
    ptrdiff_t *pp,
    double *dmin,
    double *sigma,
    double *desig,
    double *qmax,
    ptrdiff_t *nfail,
    ptrdiff_t *iter,
    ptrdiff_t *ndiv,
    ptrdiff_t *ieee,
    ptrdiff_t *ttype,
    double *dmin1,
    double *dmin2,
    double *dn,
    double *dn1,
    double *dn2,
    double *g,
    double *tau
);

/* Source: dlasq4.f */
#define dlasq4 FORTRAN_WRAPPER(dlasq4)
extern void dlasq4(
    ptrdiff_t *i0,
    ptrdiff_t *n0,
    double *z,
    ptrdiff_t *pp,
    ptrdiff_t *n0in,
    double *dmin,
    double *dmin1,
    double *dmin2,
    double *dn,
    double *dn1,
    double *dn2,
    double *tau,
    ptrdiff_t *ttype,
    double *g
);

/* Source: dlasq5.f */
#define dlasq5 FORTRAN_WRAPPER(dlasq5)
extern void dlasq5(
    ptrdiff_t *i0,
    ptrdiff_t *n0,
    double *z,
    ptrdiff_t *pp,
    double *tau,
    double *dmin,
    double *dmin1,
    double *dmin2,
    double *dn,
    double *dnm1,
    double *dnm2,
    ptrdiff_t *ieee
);

/* Source: dlasq6.f */
#define dlasq6 FORTRAN_WRAPPER(dlasq6)
extern void dlasq6(
    ptrdiff_t *i0,
    ptrdiff_t *n0,
    double *z,
    ptrdiff_t *pp,
    double *dmin,
    double *dmin1,
    double *dmin2,
    double *dn,
    double *dnm1,
    double *dnm2
);

/* Source: dlasr.f */
#define dlasr FORTRAN_WRAPPER(dlasr)
extern void dlasr(
    char   *side,
    char   *pivot,
    char   *direct,
    ptrdiff_t *m,
    ptrdiff_t *n,
    double *c,
    double *s,
    double *a,
    ptrdiff_t *lda
);

/* Source: dlasrt.f */
#define dlasrt FORTRAN_WRAPPER(dlasrt)
extern void dlasrt(
    char   *id,
    ptrdiff_t *n,
    double *d,
    ptrdiff_t *info
);

/* Source: dlassq.f */
#define dlassq FORTRAN_WRAPPER(dlassq)
extern void dlassq(
    ptrdiff_t *n,
    double *x,
    ptrdiff_t *incx,
    double *scale,
    double *sumsq
);

/* Source: dlasv2.f */
#define dlasv2 FORTRAN_WRAPPER(dlasv2)
extern void dlasv2(
    double *f,
    double *g,
    double *h,
    double *ssmin,
    double *ssmax,
    double *snr,
    double *csr,
    double *snl,
    double *csl
);

/* Source: dlaswp.f */
#define dlaswp FORTRAN_WRAPPER(dlaswp)
extern void dlaswp(
    ptrdiff_t *n,
    double *a,
    ptrdiff_t *lda,
    ptrdiff_t *k1,
    ptrdiff_t *k2,
    ptrdiff_t *ipiv,
    ptrdiff_t *incx
);

/* Source: dlasy2.f */
#define dlasy2 FORTRAN_WRAPPER(dlasy2)
extern void dlasy2(
    ptrdiff_t *ltranl,
    ptrdiff_t *ltranr,
    ptrdiff_t *isgn,
    ptrdiff_t *n1,
    ptrdiff_t *n2,
    double *tl,
    ptrdiff_t *ldtl,
    double *tr,
    ptrdiff_t *ldtr,
    double *b,
    ptrdiff_t *ldb,
    double *scale,
    double *x,
    ptrdiff_t *ldx,
    double *xnorm,
    ptrdiff_t *info
);

/* Source: dlasyf.f */
#define dlasyf FORTRAN_WRAPPER(dlasyf)
extern void dlasyf(
    char   *uplo,
    ptrdiff_t *n,
    ptrdiff_t *nb,
    ptrdiff_t *kb,
    double *a,
    ptrdiff_t *lda,
    ptrdiff_t *ipiv,
    double *w,
    ptrdiff_t *ldw,
    ptrdiff_t *info
);

/* Source: dlat2s.f */
#define dlat2s FORTRAN_WRAPPER(dlat2s)
extern void dlat2s(
    char   *uplo,
    ptrdiff_t *n,
    double *a,
    ptrdiff_t *lda,
    float  *sa,
    ptrdiff_t *ldsa,
    ptrdiff_t *info
);

/* Source: dlatbs.f */
#define dlatbs FORTRAN_WRAPPER(dlatbs)
extern void dlatbs(
    char   *uplo,
    char   *trans,
    char   *diag,
    char   *normin,
    ptrdiff_t *n,
    ptrdiff_t *kd,
    double *ab,
    ptrdiff_t *ldab,
    double *x,
    double *scale,
    double *cnorm,
    ptrdiff_t *info
);

/* Source: dlatdf.f */
#define dlatdf FORTRAN_WRAPPER(dlatdf)
extern void dlatdf(
    ptrdiff_t *ijob,
    ptrdiff_t *n,
    double *z,
    ptrdiff_t *ldz,
    double *rhs,
    double *rdsum,
    double *rdscal,
    ptrdiff_t *ipiv,
    ptrdiff_t *jpiv
);

/* Source: dlatps.f */
#define dlatps FORTRAN_WRAPPER(dlatps)
extern void dlatps(
    char   *uplo,
    char   *trans,
    char   *diag,
    char   *normin,
    ptrdiff_t *n,
    double *ap,
    double *x,
    double *scale,
    double *cnorm,
    ptrdiff_t *info
);

/* Source: dlatrd.f */
#define dlatrd FORTRAN_WRAPPER(dlatrd)
extern void dlatrd(
    char   *uplo,
    ptrdiff_t *n,
    ptrdiff_t *nb,
    double *a,
    ptrdiff_t *lda,
    double *e,
    double *tau,
    double *w,
    ptrdiff_t *ldw
);

/* Source: dlatrs.f */
#define dlatrs FORTRAN_WRAPPER(dlatrs)
extern void dlatrs(
    char   *uplo,
    char   *trans,
    char   *diag,
    char   *normin,
    ptrdiff_t *n,
    double *a,
    ptrdiff_t *lda,
    double *x,
    double *scale,
    double *cnorm,
    ptrdiff_t *info
);

/* Source: dlatrz.f */
#define dlatrz FORTRAN_WRAPPER(dlatrz)
extern void dlatrz(
    ptrdiff_t *m,
    ptrdiff_t *n,
    ptrdiff_t *l,
    double *a,
    ptrdiff_t *lda,
    double *tau,
    double *work
);

/* Source: dlatzm.f */
#define dlatzm FORTRAN_WRAPPER(dlatzm)
extern void dlatzm(
    char   *side,
    ptrdiff_t *m,
    ptrdiff_t *n,
    double *v,
    ptrdiff_t *incv,
    double *tau,
    double *c1,
    double *c2,
    ptrdiff_t *ldc,
    double *work
);

/* Source: dlauu2.f */
#define dlauu2 FORTRAN_WRAPPER(dlauu2)
extern void dlauu2(
    char   *uplo,
    ptrdiff_t *n,
    double *a,
    ptrdiff_t *lda,
    ptrdiff_t *info
);

/* Source: dlauum.f */
#define dlauum FORTRAN_WRAPPER(dlauum)
extern void dlauum(
    char   *uplo,
    ptrdiff_t *n,
    double *a,
    ptrdiff_t *lda,
    ptrdiff_t *info
);

/* Source: dopgtr.f */
#define dopgtr FORTRAN_WRAPPER(dopgtr)
extern void dopgtr(
    char   *uplo,
    ptrdiff_t *n,
    double *ap,
    double *tau,
    double *q,
    ptrdiff_t *ldq,
    double *work,
    ptrdiff_t *info
);

/* Source: dopmtr.f */
#define dopmtr FORTRAN_WRAPPER(dopmtr)
extern void dopmtr(
    char   *side,
    char   *uplo,
    char   *trans,
    ptrdiff_t *m,
    ptrdiff_t *n,
    double *ap,
    double *tau,
    double *c,
    ptrdiff_t *ldc,
    double *work,
    ptrdiff_t *info
);

/* Source: dorg2l.f */
#define dorg2l FORTRAN_WRAPPER(dorg2l)
extern void dorg2l(
    ptrdiff_t *m,
    ptrdiff_t *n,
    ptrdiff_t *k,
    double *a,
    ptrdiff_t *lda,
    double *tau,
    double *work,
    ptrdiff_t *info
);

/* Source: dorg2r.f */
#define dorg2r FORTRAN_WRAPPER(dorg2r)
extern void dorg2r(
    ptrdiff_t *m,
    ptrdiff_t *n,
    ptrdiff_t *k,
    double *a,
    ptrdiff_t *lda,
    double *tau,
    double *work,
    ptrdiff_t *info
);

/* Source: dorgbr.f */
#define dorgbr FORTRAN_WRAPPER(dorgbr)
extern void dorgbr(
    char   *vect,
    ptrdiff_t *m,
    ptrdiff_t *n,
    ptrdiff_t *k,
    double *a,
    ptrdiff_t *lda,
    double *tau,
    double *work,
    ptrdiff_t *lwork,
    ptrdiff_t *info
);

/* Source: dorghr.f */
#define dorghr FORTRAN_WRAPPER(dorghr)
extern void dorghr(
    ptrdiff_t *n,
    ptrdiff_t *ilo,
    ptrdiff_t *ihi,
    double *a,
    ptrdiff_t *lda,
    double *tau,
    double *work,
    ptrdiff_t *lwork,
    ptrdiff_t *info
);

/* Source: dorgl2.f */
#define dorgl2 FORTRAN_WRAPPER(dorgl2)
extern void dorgl2(
    ptrdiff_t *m,
    ptrdiff_t *n,
    ptrdiff_t *k,
    double *a,
    ptrdiff_t *lda,
    double *tau,
    double *work,
    ptrdiff_t *info
);

/* Source: dorglq.f */
#define dorglq FORTRAN_WRAPPER(dorglq)
extern void dorglq(
    ptrdiff_t *m,
    ptrdiff_t *n,
    ptrdiff_t *k,
    double *a,
    ptrdiff_t *lda,
    double *tau,
    double *work,
    ptrdiff_t *lwork,
    ptrdiff_t *info
);

/* Source: dorgql.f */
#define dorgql FORTRAN_WRAPPER(dorgql)
extern void dorgql(
    ptrdiff_t *m,
    ptrdiff_t *n,
    ptrdiff_t *k,
    double *a,
    ptrdiff_t *lda,
    double *tau,
    double *work,
    ptrdiff_t *lwork,
    ptrdiff_t *info
);

/* Source: dorgqr.f */
#define dorgqr FORTRAN_WRAPPER(dorgqr)
extern void dorgqr(
    ptrdiff_t *m,
    ptrdiff_t *n,
    ptrdiff_t *k,
    double *a,
    ptrdiff_t *lda,
    double *tau,
    double *work,
    ptrdiff_t *lwork,
    ptrdiff_t *info
);

/* Source: dorgr2.f */
#define dorgr2 FORTRAN_WRAPPER(dorgr2)
extern void dorgr2(
    ptrdiff_t *m,
    ptrdiff_t *n,
    ptrdiff_t *k,
    double *a,
    ptrdiff_t *lda,
    double *tau,
    double *work,
    ptrdiff_t *info
);

/* Source: dorgrq.f */
#define dorgrq FORTRAN_WRAPPER(dorgrq)
extern void dorgrq(
    ptrdiff_t *m,
    ptrdiff_t *n,
    ptrdiff_t *k,
    double *a,
    ptrdiff_t *lda,
    double *tau,
    double *work,
    ptrdiff_t *lwork,
    ptrdiff_t *info
);

/* Source: dorgtr.f */
#define dorgtr FORTRAN_WRAPPER(dorgtr)
extern void dorgtr(
    char   *uplo,
    ptrdiff_t *n,
    double *a,
    ptrdiff_t *lda,
    double *tau,
    double *work,
    ptrdiff_t *lwork,
    ptrdiff_t *info
);

/* Source: dorm2l.f */
#define dorm2l FORTRAN_WRAPPER(dorm2l)
extern void dorm2l(
    char   *side,
    char   *trans,
    ptrdiff_t *m,
    ptrdiff_t *n,
    ptrdiff_t *k,
    double *a,
    ptrdiff_t *lda,
    double *tau,
    double *c,
    ptrdiff_t *ldc,
    double *work,
    ptrdiff_t *info
);

/* Source: dorm2r.f */
#define dorm2r FORTRAN_WRAPPER(dorm2r)
extern void dorm2r(
    char   *side,
    char   *trans,
    ptrdiff_t *m,
    ptrdiff_t *n,
    ptrdiff_t *k,
    double *a,
    ptrdiff_t *lda,
    double *tau,
    double *c,
    ptrdiff_t *ldc,
    double *work,
    ptrdiff_t *info
);

/* Source: dormbr.f */
#define dormbr FORTRAN_WRAPPER(dormbr)
extern void dormbr(
    char   *vect,
    char   *side,
    char   *trans,
    ptrdiff_t *m,
    ptrdiff_t *n,
    ptrdiff_t *k,
    double *a,
    ptrdiff_t *lda,
    double *tau,
    double *c,
    ptrdiff_t *ldc,
    double *work,
    ptrdiff_t *lwork,
    ptrdiff_t *info
);

/* Source: dormhr.f */
#define dormhr FORTRAN_WRAPPER(dormhr)
extern void dormhr(
    char   *side,
    char   *trans,
    ptrdiff_t *m,
    ptrdiff_t *n,
    ptrdiff_t *ilo,
    ptrdiff_t *ihi,
    double *a,
    ptrdiff_t *lda,
    double *tau,
    double *c,
    ptrdiff_t *ldc,
    double *work,
    ptrdiff_t *lwork,
    ptrdiff_t *info
);

/* Source: dorml2.f */
#define dorml2 FORTRAN_WRAPPER(dorml2)
extern void dorml2(
    char   *side,
    char   *trans,
    ptrdiff_t *m,
    ptrdiff_t *n,
    ptrdiff_t *k,
    double *a,
    ptrdiff_t *lda,
    double *tau,
    double *c,
    ptrdiff_t *ldc,
    double *work,
    ptrdiff_t *info
);

/* Source: dormlq.f */
#define dormlq FORTRAN_WRAPPER(dormlq)
extern void dormlq(
    char   *side,
    char   *trans,
    ptrdiff_t *m,
    ptrdiff_t *n,
    ptrdiff_t *k,
    double *a,
    ptrdiff_t *lda,
    double *tau,
    double *c,
    ptrdiff_t *ldc,
    double *work,
    ptrdiff_t *lwork,
    ptrdiff_t *info
);

/* Source: dormql.f */
#define dormql FORTRAN_WRAPPER(dormql)
extern void dormql(
    char   *side,
    char   *trans,
    ptrdiff_t *m,
    ptrdiff_t *n,
    ptrdiff_t *k,
    double *a,
    ptrdiff_t *lda,
    double *tau,
    double *c,
    ptrdiff_t *ldc,
    double *work,
    ptrdiff_t *lwork,
    ptrdiff_t *info
);

/* Source: dormqr.f */
#define dormqr FORTRAN_WRAPPER(dormqr)
extern void dormqr(
    char   *side,
    char   *trans,
    ptrdiff_t *m,
    ptrdiff_t *n,
    ptrdiff_t *k,
    double *a,
    ptrdiff_t *lda,
    double *tau,
    double *c,
    ptrdiff_t *ldc,
    double *work,
    ptrdiff_t *lwork,
    ptrdiff_t *info
);

/* Source: dormr2.f */
#define dormr2 FORTRAN_WRAPPER(dormr2)
extern void dormr2(
    char   *side,
    char   *trans,
    ptrdiff_t *m,
    ptrdiff_t *n,
    ptrdiff_t *k,
    double *a,
    ptrdiff_t *lda,
    double *tau,
    double *c,
    ptrdiff_t *ldc,
    double *work,
    ptrdiff_t *info
);

/* Source: dormr3.f */
#define dormr3 FORTRAN_WRAPPER(dormr3)
extern void dormr3(
    char   *side,
    char   *trans,
    ptrdiff_t *m,
    ptrdiff_t *n,
    ptrdiff_t *k,
    ptrdiff_t *l,
    double *a,
    ptrdiff_t *lda,
    double *tau,
    double *c,
    ptrdiff_t *ldc,
    double *work,
    ptrdiff_t *info
);

/* Source: dormrq.f */
#define dormrq FORTRAN_WRAPPER(dormrq)
extern void dormrq(
    char   *side,
    char   *trans,
    ptrdiff_t *m,
    ptrdiff_t *n,
    ptrdiff_t *k,
    double *a,
    ptrdiff_t *lda,
    double *tau,
    double *c,
    ptrdiff_t *ldc,
    double *work,
    ptrdiff_t *lwork,
    ptrdiff_t *info
);

/* Source: dormrz.f */
#define dormrz FORTRAN_WRAPPER(dormrz)
extern void dormrz(
    char   *side,
    char   *trans,
    ptrdiff_t *m,
    ptrdiff_t *n,
    ptrdiff_t *k,
    ptrdiff_t *l,
    double *a,
    ptrdiff_t *lda,
    double *tau,
    double *c,
    ptrdiff_t *ldc,
    double *work,
    ptrdiff_t *lwork,
    ptrdiff_t *info
);

/* Source: dormtr.f */
#define dormtr FORTRAN_WRAPPER(dormtr)
extern void dormtr(
    char   *side,
    char   *uplo,
    char   *trans,
    ptrdiff_t *m,
    ptrdiff_t *n,
    double *a,
    ptrdiff_t *lda,
    double *tau,
    double *c,
    ptrdiff_t *ldc,
    double *work,
    ptrdiff_t *lwork,
    ptrdiff_t *info
);

/* Source: dpbcon.f */
#define dpbcon FORTRAN_WRAPPER(dpbcon)
extern void dpbcon(
    char   *uplo,
    ptrdiff_t *n,
    ptrdiff_t *kd,
    double *ab,
    ptrdiff_t *ldab,
    double *anorm,
    double *rcond,
    double *work,
    ptrdiff_t *iwork,
    ptrdiff_t *info
);

/* Source: dpbequ.f */
#define dpbequ FORTRAN_WRAPPER(dpbequ)
extern void dpbequ(
    char   *uplo,
    ptrdiff_t *n,
    ptrdiff_t *kd,
    double *ab,
    ptrdiff_t *ldab,
    double *s,
    double *scond,
    double *amax,
    ptrdiff_t *info
);

/* Source: dpbrfs.f */
#define dpbrfs FORTRAN_WRAPPER(dpbrfs)
extern void dpbrfs(
    char   *uplo,
    ptrdiff_t *n,
    ptrdiff_t *kd,
    ptrdiff_t *nrhs,
    double *ab,
    ptrdiff_t *ldab,
    double *afb,
    ptrdiff_t *ldafb,
    double *b,
    ptrdiff_t *ldb,
    double *x,
    ptrdiff_t *ldx,
    double *ferr,
    double *berr,
    double *work,
    ptrdiff_t *iwork,
    ptrdiff_t *info
);

/* Source: dpbstf.f */
#define dpbstf FORTRAN_WRAPPER(dpbstf)
extern void dpbstf(
    char   *uplo,
    ptrdiff_t *n,
    ptrdiff_t *kd,
    double *ab,
    ptrdiff_t *ldab,
    ptrdiff_t *info
);

/* Source: dpbsv.f */
#define dpbsv FORTRAN_WRAPPER(dpbsv)
extern void dpbsv(
    char   *uplo,
    ptrdiff_t *n,
    ptrdiff_t *kd,
    ptrdiff_t *nrhs,
    double *ab,
    ptrdiff_t *ldab,
    double *b,
    ptrdiff_t *ldb,
    ptrdiff_t *info
);

/* Source: dpbsvx.f */
#define dpbsvx FORTRAN_WRAPPER(dpbsvx)
extern void dpbsvx(
    char   *fact,
    char   *uplo,
    ptrdiff_t *n,
    ptrdiff_t *kd,
    ptrdiff_t *nrhs,
    double *ab,
    ptrdiff_t *ldab,
    double *afb,
    ptrdiff_t *ldafb,
    char   *equed,
    double *s,
    double *b,
    ptrdiff_t *ldb,
    double *x,
    ptrdiff_t *ldx,
    double *rcond,
    double *ferr,
    double *berr,
    double *work,
    ptrdiff_t *iwork,
    ptrdiff_t *info
);

/* Source: dpbtf2.f */
#define dpbtf2 FORTRAN_WRAPPER(dpbtf2)
extern void dpbtf2(
    char   *uplo,
    ptrdiff_t *n,
    ptrdiff_t *kd,
    double *ab,
    ptrdiff_t *ldab,
    ptrdiff_t *info
);

/* Source: dpbtrf.f */
#define dpbtrf FORTRAN_WRAPPER(dpbtrf)
extern void dpbtrf(
    char   *uplo,
    ptrdiff_t *n,
    ptrdiff_t *kd,
    double *ab,
    ptrdiff_t *ldab,
    ptrdiff_t *info
);

/* Source: dpbtrs.f */
#define dpbtrs FORTRAN_WRAPPER(dpbtrs)
extern void dpbtrs(
    char   *uplo,
    ptrdiff_t *n,
    ptrdiff_t *kd,
    ptrdiff_t *nrhs,
    double *ab,
    ptrdiff_t *ldab,
    double *b,
    ptrdiff_t *ldb,
    ptrdiff_t *info
);

/* Source: dpftrf.f */
#define dpftrf FORTRAN_WRAPPER(dpftrf)
extern void dpftrf(
    char   *transr,
    char   *uplo,
    ptrdiff_t *n,
    double *a,
    ptrdiff_t *info
);

/* Source: dpftri.f */
#define dpftri FORTRAN_WRAPPER(dpftri)
extern void dpftri(
    char   *transr,
    char   *uplo,
    ptrdiff_t *n,
    double *a,
    ptrdiff_t *info
);

/* Source: dpftrs.f */
#define dpftrs FORTRAN_WRAPPER(dpftrs)
extern void dpftrs(
    char   *transr,
    char   *uplo,
    ptrdiff_t *n,
    ptrdiff_t *nrhs,
    double *a,
    double *b,
    ptrdiff_t *ldb,
    ptrdiff_t *info
);

/* Source: dpocon.f */
#define dpocon FORTRAN_WRAPPER(dpocon)
extern void dpocon(
    char   *uplo,
    ptrdiff_t *n,
    double *a,
    ptrdiff_t *lda,
    double *anorm,
    double *rcond,
    double *work,
    ptrdiff_t *iwork,
    ptrdiff_t *info
);

/* Source: dpoequ.f */
#define dpoequ FORTRAN_WRAPPER(dpoequ)
extern void dpoequ(
    ptrdiff_t *n,
    double *a,
    ptrdiff_t *lda,
    double *s,
    double *scond,
    double *amax,
    ptrdiff_t *info
);

/* Source: dpoequb.f */
#define dpoequb FORTRAN_WRAPPER(dpoequb)
extern void dpoequb(
    ptrdiff_t *n,
    double *a,
    ptrdiff_t *lda,
    double *s,
    double *scond,
    double *amax,
    ptrdiff_t *info
);

/* Source: dporfs.f */
#define dporfs FORTRAN_WRAPPER(dporfs)
extern void dporfs(
    char   *uplo,
    ptrdiff_t *n,
    ptrdiff_t *nrhs,
    double *a,
    ptrdiff_t *lda,
    double *af,
    ptrdiff_t *ldaf,
    double *b,
    ptrdiff_t *ldb,
    double *x,
    ptrdiff_t *ldx,
    double *ferr,
    double *berr,
    double *work,
    ptrdiff_t *iwork,
    ptrdiff_t *info
);

/* Source: dposv.f */
#define dposv FORTRAN_WRAPPER(dposv)
extern void dposv(
    char   *uplo,
    ptrdiff_t *n,
    ptrdiff_t *nrhs,
    double *a,
    ptrdiff_t *lda,
    double *b,
    ptrdiff_t *ldb,
    ptrdiff_t *info
);

/* Source: dposvx.f */
#define dposvx FORTRAN_WRAPPER(dposvx)
extern void dposvx(
    char   *fact,
    char   *uplo,
    ptrdiff_t *n,
    ptrdiff_t *nrhs,
    double *a,
    ptrdiff_t *lda,
    double *af,
    ptrdiff_t *ldaf,
    char   *equed,
    double *s,
    double *b,
    ptrdiff_t *ldb,
    double *x,
    ptrdiff_t *ldx,
    double *rcond,
    double *ferr,
    double *berr,
    double *work,
    ptrdiff_t *iwork,
    ptrdiff_t *info
);

/* Source: dpotf2.f */
#define dpotf2 FORTRAN_WRAPPER(dpotf2)
extern void dpotf2(
    char   *uplo,
    ptrdiff_t *n,
    double *a,
    ptrdiff_t *lda,
    ptrdiff_t *info
);

/* Source: dpotrf.f */
#define dpotrf FORTRAN_WRAPPER(dpotrf)
extern void dpotrf(
    char   *uplo,
    ptrdiff_t *n,
    double *a,
    ptrdiff_t *lda,
    ptrdiff_t *info
);

/* Source: dpotri.f */
#define dpotri FORTRAN_WRAPPER(dpotri)
extern void dpotri(
    char   *uplo,
    ptrdiff_t *n,
    double *a,
    ptrdiff_t *lda,
    ptrdiff_t *info
);

/* Source: dpotrs.f */
#define dpotrs FORTRAN_WRAPPER(dpotrs)
extern void dpotrs(
    char   *uplo,
    ptrdiff_t *n,
    ptrdiff_t *nrhs,
    double *a,
    ptrdiff_t *lda,
    double *b,
    ptrdiff_t *ldb,
    ptrdiff_t *info
);

/* Source: dppcon.f */
#define dppcon FORTRAN_WRAPPER(dppcon)
extern void dppcon(
    char   *uplo,
    ptrdiff_t *n,
    double *ap,
    double *anorm,
    double *rcond,
    double *work,
    ptrdiff_t *iwork,
    ptrdiff_t *info
);

/* Source: dppequ.f */
#define dppequ FORTRAN_WRAPPER(dppequ)
extern void dppequ(
    char   *uplo,
    ptrdiff_t *n,
    double *ap,
    double *s,
    double *scond,
    double *amax,
    ptrdiff_t *info
);

/* Source: dpprfs.f */
#define dpprfs FORTRAN_WRAPPER(dpprfs)
extern void dpprfs(
    char   *uplo,
    ptrdiff_t *n,
    ptrdiff_t *nrhs,
    double *ap,
    double *afp,
    double *b,
    ptrdiff_t *ldb,
    double *x,
    ptrdiff_t *ldx,
    double *ferr,
    double *berr,
    double *work,
    ptrdiff_t *iwork,
    ptrdiff_t *info
);

/* Source: dppsv.f */
#define dppsv FORTRAN_WRAPPER(dppsv)
extern void dppsv(
    char   *uplo,
    ptrdiff_t *n,
    ptrdiff_t *nrhs,
    double *ap,
    double *b,
    ptrdiff_t *ldb,
    ptrdiff_t *info
);

/* Source: dppsvx.f */
#define dppsvx FORTRAN_WRAPPER(dppsvx)
extern void dppsvx(
    char   *fact,
    char   *uplo,
    ptrdiff_t *n,
    ptrdiff_t *nrhs,
    double *ap,
    double *afp,
    char   *equed,
    double *s,
    double *b,
    ptrdiff_t *ldb,
    double *x,
    ptrdiff_t *ldx,
    double *rcond,
    double *ferr,
    double *berr,
    double *work,
    ptrdiff_t *iwork,
    ptrdiff_t *info
);

/* Source: dpptrf.f */
#define dpptrf FORTRAN_WRAPPER(dpptrf)
extern void dpptrf(
    char   *uplo,
    ptrdiff_t *n,
    double *ap,
    ptrdiff_t *info
);

/* Source: dpptri.f */
#define dpptri FORTRAN_WRAPPER(dpptri)
extern void dpptri(
    char   *uplo,
    ptrdiff_t *n,
    double *ap,
    ptrdiff_t *info
);

/* Source: dpptrs.f */
#define dpptrs FORTRAN_WRAPPER(dpptrs)
extern void dpptrs(
    char   *uplo,
    ptrdiff_t *n,
    ptrdiff_t *nrhs,
    double *ap,
    double *b,
    ptrdiff_t *ldb,
    ptrdiff_t *info
);

/* Source: dpstf2.f */
#define dpstf2 FORTRAN_WRAPPER(dpstf2)
extern void dpstf2(
    char   *uplo,
    ptrdiff_t *n,
    double *a,
    ptrdiff_t *lda,
    ptrdiff_t *piv,
    ptrdiff_t *rank,
    double *tol,
    double *work,
    ptrdiff_t *info
);

/* Source: dpstrf.f */
#define dpstrf FORTRAN_WRAPPER(dpstrf)
extern void dpstrf(
    char   *uplo,
    ptrdiff_t *n,
    double *a,
    ptrdiff_t *lda,
    ptrdiff_t *piv,
    ptrdiff_t *rank,
    double *tol,
    double *work,
    ptrdiff_t *info
);

/* Source: dptcon.f */
#define dptcon FORTRAN_WRAPPER(dptcon)
extern void dptcon(
    ptrdiff_t *n,
    double *d,
    double *e,
    double *anorm,
    double *rcond,
    double *work,
    ptrdiff_t *info
);

/* Source: dpteqr.f */
#define dpteqr FORTRAN_WRAPPER(dpteqr)
extern void dpteqr(
    char   *compz,
    ptrdiff_t *n,
    double *d,
    double *e,
    double *z,
    ptrdiff_t *ldz,
    double *work,
    ptrdiff_t *info
);

/* Source: dptrfs.f */
#define dptrfs FORTRAN_WRAPPER(dptrfs)
extern void dptrfs(
    ptrdiff_t *n,
    ptrdiff_t *nrhs,
    double *d,
    double *e,
    double *df,
    double *ef,
    double *b,
    ptrdiff_t *ldb,
    double *x,
    ptrdiff_t *ldx,
    double *ferr,
    double *berr,
    double *work,
    ptrdiff_t *info
);

/* Source: dptsv.f */
#define dptsv FORTRAN_WRAPPER(dptsv)
extern void dptsv(
    ptrdiff_t *n,
    ptrdiff_t *nrhs,
    double *d,
    double *e,
    double *b,
    ptrdiff_t *ldb,
    ptrdiff_t *info
);

/* Source: dptsvx.f */
#define dptsvx FORTRAN_WRAPPER(dptsvx)
extern void dptsvx(
    char   *fact,
    ptrdiff_t *n,
    ptrdiff_t *nrhs,
    double *d,
    double *e,
    double *df,
    double *ef,
    double *b,
    ptrdiff_t *ldb,
    double *x,
    ptrdiff_t *ldx,
    double *rcond,
    double *ferr,
    double *berr,
    double *work,
    ptrdiff_t *info
);

/* Source: dpttrf.f */
#define dpttrf FORTRAN_WRAPPER(dpttrf)
extern void dpttrf(
    ptrdiff_t *n,
    double *d,
    double *e,
    ptrdiff_t *info
);

/* Source: dpttrs.f */
#define dpttrs FORTRAN_WRAPPER(dpttrs)
extern void dpttrs(
    ptrdiff_t *n,
    ptrdiff_t *nrhs,
    double *d,
    double *e,
    double *b,
    ptrdiff_t *ldb,
    ptrdiff_t *info
);

/* Source: dptts2.f */
#define dptts2 FORTRAN_WRAPPER(dptts2)
extern void dptts2(
    ptrdiff_t *n,
    ptrdiff_t *nrhs,
    double *d,
    double *e,
    double *b,
    ptrdiff_t *ldb
);

/* Source: drscl.f */
#define drscl FORTRAN_WRAPPER(drscl)
extern void drscl(
    ptrdiff_t *n,
    double *sa,
    double *sx,
    ptrdiff_t *incx
);

/* Source: dsbev.f */
#define dsbev FORTRAN_WRAPPER(dsbev)
extern void dsbev(
    char   *jobz,
    char   *uplo,
    ptrdiff_t *n,
    ptrdiff_t *kd,
    double *ab,
    ptrdiff_t *ldab,
    double *w,
    double *z,
    ptrdiff_t *ldz,
    double *work,
    ptrdiff_t *info
);

/* Source: dsbevd.f */
#define dsbevd FORTRAN_WRAPPER(dsbevd)
extern void dsbevd(
    char   *jobz,
    char   *uplo,
    ptrdiff_t *n,
    ptrdiff_t *kd,
    double *ab,
    ptrdiff_t *ldab,
    double *w,
    double *z,
    ptrdiff_t *ldz,
    double *work,
    ptrdiff_t *lwork,
    ptrdiff_t *iwork,
    ptrdiff_t *liwork,
    ptrdiff_t *info
);

/* Source: dsbevx.f */
#define dsbevx FORTRAN_WRAPPER(dsbevx)
extern void dsbevx(
    char   *jobz,
    char   *range,
    char   *uplo,
    ptrdiff_t *n,
    ptrdiff_t *kd,
    double *ab,
    ptrdiff_t *ldab,
    double *q,
    ptrdiff_t *ldq,
    double *vl,
    double *vu,
    ptrdiff_t *il,
    ptrdiff_t *iu,
    double *abstol,
    ptrdiff_t *m,
    double *w,
    double *z,
    ptrdiff_t *ldz,
    double *work,
    ptrdiff_t *iwork,
    ptrdiff_t *ifail,
    ptrdiff_t *info
);

/* Source: dsbgst.f */
#define dsbgst FORTRAN_WRAPPER(dsbgst)
extern void dsbgst(
    char   *vect,
    char   *uplo,
    ptrdiff_t *n,
    ptrdiff_t *ka,
    ptrdiff_t *kb,
    double *ab,
    ptrdiff_t *ldab,
    double *bb,
    ptrdiff_t *ldbb,
    double *x,
    ptrdiff_t *ldx,
    double *work,
    ptrdiff_t *info
);

/* Source: dsbgv.f */
#define dsbgv FORTRAN_WRAPPER(dsbgv)
extern void dsbgv(
    char   *jobz,
    char   *uplo,
    ptrdiff_t *n,
    ptrdiff_t *ka,
    ptrdiff_t *kb,
    double *ab,
    ptrdiff_t *ldab,
    double *bb,
    ptrdiff_t *ldbb,
    double *w,
    double *z,
    ptrdiff_t *ldz,
    double *work,
    ptrdiff_t *info
);

/* Source: dsbgvd.f */
#define dsbgvd FORTRAN_WRAPPER(dsbgvd)
extern void dsbgvd(
    char   *jobz,
    char   *uplo,
    ptrdiff_t *n,
    ptrdiff_t *ka,
    ptrdiff_t *kb,
    double *ab,
    ptrdiff_t *ldab,
    double *bb,
    ptrdiff_t *ldbb,
    double *w,
    double *z,
    ptrdiff_t *ldz,
    double *work,
    ptrdiff_t *lwork,
    ptrdiff_t *iwork,
    ptrdiff_t *liwork,
    ptrdiff_t *info
);

/* Source: dsbgvx.f */
#define dsbgvx FORTRAN_WRAPPER(dsbgvx)
extern void dsbgvx(
    char   *jobz,
    char   *range,
    char   *uplo,
    ptrdiff_t *n,
    ptrdiff_t *ka,
    ptrdiff_t *kb,
    double *ab,
    ptrdiff_t *ldab,
    double *bb,
    ptrdiff_t *ldbb,
    double *q,
    ptrdiff_t *ldq,
    double *vl,
    double *vu,
    ptrdiff_t *il,
    ptrdiff_t *iu,
    double *abstol,
    ptrdiff_t *m,
    double *w,
    double *z,
    ptrdiff_t *ldz,
    double *work,
    ptrdiff_t *iwork,
    ptrdiff_t *ifail,
    ptrdiff_t *info
);

/* Source: dsbtrd.f */
#define dsbtrd FORTRAN_WRAPPER(dsbtrd)
extern void dsbtrd(
    char   *vect,
    char   *uplo,
    ptrdiff_t *n,
    ptrdiff_t *kd,
    double *ab,
    ptrdiff_t *ldab,
    double *d,
    double *e,
    double *q,
    ptrdiff_t *ldq,
    double *work,
    ptrdiff_t *info
);

/* Source: dsfrk.f */
#define dsfrk FORTRAN_WRAPPER(dsfrk)
extern void dsfrk(
    char   *transr,
    char   *uplo,
    char   *trans,
    ptrdiff_t *n,
    ptrdiff_t *k,
    double *alpha,
    double *a,
    ptrdiff_t *lda,
    double *beta,
    double *c
);

/* Source: dsgesv.f */
#define dsgesv FORTRAN_WRAPPER(dsgesv)
extern void dsgesv(
    ptrdiff_t *n,
    ptrdiff_t *nrhs,
    double *a,
    ptrdiff_t *lda,
    ptrdiff_t *ipiv,
    double *b,
    ptrdiff_t *ldb,
    double *x,
    ptrdiff_t *ldx,
    double *work,
    float  *swork,
    ptrdiff_t *iter,
    ptrdiff_t *info
);
```
